    // Detect ON/OFF state change
    IF aUnits[i].bPresVal <> aPrevState[i] THEN
        // --------------------------------------------------------
        // (a) Send TwinCAT message as before
        // --------------------------------------------------------
        IF aUnits[i].bPresVal THEN
            sMsgText := CONCAT(stUnit.sUnitName, ' is Turned ON');
        ELSE
            sMsgText := CONCAT(stUnit.sUnitName, ' is Turned OFF');
        END_IF

        fbMsg.CreateEx(TC_EVENTS.UnitPowerStatus.EventPowerStatus, 0);
        fbMsg.ipArguments.AddString(sMsgText);
        fbMsg.Send(0);

        // --------------------------------------------------------
        // (b) Push event to global CSV queue (for P_CSVWrite_TextMode)
        // --------------------------------------------------------
        IF g_iCount < g_CSV_BUF_SIZE THEN
            g_aUnitName[g_iWriteIdx] := stUnit.sUnitName;
            g_aState[g_iWriteIdx]    := aUnits[i].bPresVal;
            g_iWriteIdx := g_iWriteIdx + 1;
            IF g_iWriteIdx > g_CSV_BUF_SIZE THEN g_iWriteIdx := 1; END_IF
            g_iCount := g_iCount + 1;
        END_IF

        // --------------------------------------------------------
        // (c) Update previous state
        // --------------------------------------------------------
        aPrevState[i] := aUnits[i].bPresVal;
    END_IF
END_FOR

// ------------------------------------------------------------
// Optional debug info
// ------------------------------------------------------------
sDebug := CONCAT('Queued=', INT_TO_STRING(g_iCount));

END_FUNCTION_BLOCK

// ---- POUs/FB_EventLogger/FB_EventF28.TcPOU
FUNCTION_BLOCK FB_EventF28
VAR_INPUT
	FB_Bacnet : FB_BACnet_DAIKIN_MasterStation_III_No_7;
END_VAR
VAR_OUTPUT
	sDebug : STRING(200);
END_VAR
VAR
	fbMsg : FB_TcMessage;
	aUnits : ARRAY[1..23] OF AC_Unit_Status;
	stUnit   : AC_Unit_Status;
	i: INT;
	sMsgText: STRING;

END_VAR
VAR RETAIN
	aPrevState : ARRAY[1..23] OF BOOL := [FALSE(*23*)];
END_VAR


aUnits[1].bPresVal := FB_Bacnet.StartStopStatus_064.bPresVal;
aUnits[1].sUnitName := 'F28-A1 (1-00)';
aUnits[2].bPresVal := FB_Bacnet.StartStopStatus_065.bPresVal;
aUnits[2].sUnitName := 'F28-A2 (1-01)';
aUnits[3].bPresVal := FB_Bacnet.StartStopStatus_066.bPresVal;
aUnits[3].sUnitName := 'F28-A3 (1-02)';
aUnits[4].bPresVal := FB_Bacnet.StartStopStatus_067.bPresVal;
aUnits[4].sUnitName := 'F28-A4 (1-03)';
aUnits[5].bPresVal := FB_Bacnet.StartStopStatus_068.bPresVal;
aUnits[5].sUnitName := 'F28-B1 (1-04)';
aUnits[6].bPresVal := FB_Bacnet.StartStopStatus_069.bPresVal;
aUnits[6].sUnitName := 'F28-B2 (1-05)';
aUnits[7].bPresVal := FB_Bacnet.StartStopStatus_070.bPresVal;
aUnits[7].sUnitName := 'F28-C1 (1-06)';
aUnits[8].bPresVal := FB_Bacnet.StartStopStatus_071.bPresVal;
aUnits[8].sUnitName := 'F28-C2 (1-07)';
aUnits[9].bPresVal := FB_Bacnet.StartStopStatus_072.bPresVal;
aUnits[9].sUnitName := 'F28-D1 (1-08)';
aUnits[10].bPresVal := FB_Bacnet.StartStopStatus_073.bPresVal;
aUnits[10].sUnitName := 'F28-D2 (1-09)';
aUnits[11].bPresVal := FB_Bacnet.StartStopStatus_074.bPresVal;
aUnits[11].sUnitName := 'F28-D3 (1-10)';
aUnits[12].bPresVal := FB_Bacnet.StartStopStatus_075.bPresVal;
aUnits[12].sUnitName := 'F28-D4 (1-11)';
aUnits[13].bPresVal := FB_Bacnet.StartStopStatus_076.bPresVal;
aUnits[13].sUnitName := 'F28-E1 (1-12)';
aUnits[14].bPresVal := FB_Bacnet.StartStopStatus_077.bPresVal;
aUnits[14].sUnitName := 'F28-E2 (1-13)';
aUnits[15].bPresVal := FB_Bacnet.StartStopStatus_078.bPresVal;
aUnits[15].sUnitName := 'F28-E3 (1-14)';
aUnits[16].bPresVal := FB_Bacnet.StartStopStatus_079.bPresVal;
aUnits[16].sUnitName := 'F28-F1 (1-15)';
aUnits[17].bPresVal := FB_Bacnet.StartStopStatus_080.bPresVal;
aUnits[17].sUnitName := 'F28-F2 (2-00)';
aUnits[18].bPresVal := FB_Bacnet.StartStopStatus_081.bPresVal;
aUnits[18].sUnitName := 'F28-G1 (2-01)';
aUnits[19].bPresVal := FB_Bacnet.StartStopStatus_082.bPresVal;
aUnits[19].sUnitName := 'F28-G2 (2-02)';
aUnits[20].bPresVal := FB_Bacnet.StartStopStatus_083.bPresVal;
aUnits[20].sUnitName := 'F28-H (2-03)';
aUnits[21].bPresVal := FB_Bacnet.StartStopStatus_112.bPresVal;
aUnits[21].sUnitName := 'F28-IT-1 (4-00)';
aUnits[22].bPresVal := FB_Bacnet.StartStopStatus_241.bPresVal;
aUnits[22].sUnitName := 'F28-IT-2 (4-01)';
aUnits[23].bPresVal := FB_Bacnet.StartStopStatus_225.bPresVal;
aUnits[23].sUnitName := 'F28-Lobi (3-01)';

FOR i := 1 TO 23 DO
    stUnit := aUnits[i];

    // Detect ON/OFF state change
    IF aUnits[i].bPresVal <> aPrevState[i] THEN
        // --------------------------------------------------------
        // (a) Send TwinCAT message as before
        // --------------------------------------------------------
        IF aUnits[i].bPresVal THEN
            sMsgText := CONCAT(stUnit.sUnitName, ' is Turned ON');
        ELSE
            sMsgText := CONCAT(stUnit.sUnitName, ' is Turned OFF');
        END_IF

        fbMsg.CreateEx(TC_EVENTS.UnitPowerStatus.EventPowerStatus, 0);
        fbMsg.ipArguments.AddString(sMsgText);
        fbMsg.Send(0);

        // --------------------------------------------------------
        // (b) Push event to global CSV queue (for P_CSVWrite_TextMode)
        // --------------------------------------------------------
        IF g_iCount < g_CSV_BUF_SIZE THEN
            g_aUnitName[g_iWriteIdx] := stUnit.sUnitName;
            g_aState[g_iWriteIdx]    := aUnits[i].bPresVal;
            g_iWriteIdx := g_iWriteIdx + 1;
            IF g_iWriteIdx > g_CSV_BUF_SIZE THEN g_iWriteIdx := 1; END_IF
            g_iCount := g_iCount + 1;
        END_IF

        // --------------------------------------------------------
        // (c) Update previous state
        // --------------------------------------------------------
        aPrevState[i] := aUnits[i].bPresVal;
    END_IF
END_FOR

// ------------------------------------------------------------
// Optional debug info
// ------------------------------------------------------------
sDebug := CONCAT('Queued=', INT_TO_STRING(g_iCount));

END_FUNCTION_BLOCK

// ---- POUs/FB_EventLogger/FB_EventF29.TcPOU
FUNCTION_BLOCK FB_EventF29
VAR_INPUT
	FB_Bacnet : FB_BACnet_DAIKIN_MasterStation_III_No_7;
END_VAR
VAR_OUTPUT
	sDebug : STRING(200);
END_VAR
VAR
	fbMsg : FB_TcMessage;
	aUnits : ARRAY[1..23] OF AC_Unit_Status;
	stUnit   : AC_Unit_Status;
	i: INT;
	sMsgText: STRING;

END_VAR
VAR RETAIN
	aPrevState : ARRAY[1..23] OF BOOL := [FALSE(*23*)];
END_VAR


aUnits[1].bPresVal := FB_Bacnet.StartStopStatus_128.bPresVal;
aUnits[1].sUnitName := 'F29-A1 (1-00)';
aUnits[2].bPresVal := FB_Bacnet.StartStopStatus_129.bPresVal;
aUnits[2].sUnitName := 'F29-A2 (1-01)';
aUnits[3].bPresVal := FB_Bacnet.StartStopStatus_130.bPresVal;
aUnits[3].sUnitName := 'F29-A3 (1-02)';
aUnits[4].bPresVal := FB_Bacnet.StartStopStatus_131.bPresVal;
aUnits[4].sUnitName := 'F29-A4 (1-03)';
aUnits[5].bPresVal := FB_Bacnet.StartStopStatus_132.bPresVal;
aUnits[5].sUnitName := 'F29-B1 (1-04)';
aUnits[6].bPresVal := FB_Bacnet.StartStopStatus_133.bPresVal;
aUnits[6].sUnitName := 'F29-B2 (1-05)';
aUnits[7].bPresVal := FB_Bacnet.StartStopStatus_134.bPresVal;
aUnits[7].sUnitName := 'F29-C1 (1-06)';
aUnits[8].bPresVal := FB_Bacnet.StartStopStatus_135.bPresVal;
aUnits[8].sUnitName := 'F29-C2 (1-07)';
aUnits[9].bPresVal := FB_Bacnet.StartStopStatus_136.bPresVal;
aUnits[9].sUnitName := 'F29-D1 (1-08)';
aUnits[10].bPresVal := FB_Bacnet.StartStopStatus_137.bPresVal;
aUnits[10].sUnitName := 'F29-D2 (1-09)';
aUnits[11].bPresVal := FB_Bacnet.StartStopStatus_138.bPresVal;
aUnits[11].sUnitName := 'F29-D3 (1-10)';
aUnits[12].bPresVal := FB_Bacnet.StartStopStatus_139.bPresVal;
aUnits[12].sUnitName := 'F29-D4 (1-11)';
aUnits[13].bPresVal := FB_Bacnet.StartStopStatus_140.bPresVal;
aUnits[13].sUnitName := 'F29-E1 (1-12)';
aUnits[14].bPresVal := FB_Bacnet.StartStopStatus_141.bPresVal;
aUnits[14].sUnitName := 'F29-E2 (1-13)';
aUnits[15].bPresVal := FB_Bacnet.StartStopStatus_142.bPresVal;
aUnits[15].sUnitName := 'F29-E3 (1-14)';
aUnits[16].bPresVal := FB_Bacnet.StartStopStatus_143.bPresVal;
aUnits[16].sUnitName := 'F29-F1 (1-15)';
aUnits[17].bPresVal := FB_Bacnet.StartStopStatus_144.bPresVal;
aUnits[17].sUnitName := 'F29-F2 (2-00)';
aUnits[18].bPresVal := FB_Bacnet.StartStopStatus_145.bPresVal;
aUnits[18].sUnitName := 'F29-G1 (2-01)';
aUnits[19].bPresVal := FB_Bacnet.StartStopStatus_146.bPresVal;
aUnits[19].sUnitName := 'F29-G2 (2-02)';
aUnits[20].bPresVal := FB_Bacnet.StartStopStatus_147.bPresVal;
aUnits[20].sUnitName := 'F29-H (2-03)';
aUnits[21].bPresVal := FB_Bacnet.StartStopStatus_148.bPresVal;
aUnits[21].sUnitName := 'F29-LMR-1 (2-04)';
aUnits[22].bPresVal := FB_Bacnet.StartStopStatus_149.bPresVal;
aUnits[22].sUnitName := 'F29-LMR-2 (2-05)';
aUnits[23].bPresVal := FB_Bacnet.StartStopStatus_226.bPresVal;
aUnits[23].sUnitName := 'F29-Lobi (3-02)';

FOR i := 1 TO 23 DO
    stUnit := aUnits[i];

    // Detect ON/OFF state change
    IF aUnits[i].bPresVal <> aPrevState[i] THEN
        // --------------------------------------------------------
        // (a) Send TwinCAT message as before
        // --------------------------------------------------------
        IF aUnits[i].bPresVal THEN
            sMsgText := CONCAT(stUnit.sUnitName, ' is Turned ON');
        ELSE
            sMsgText := CONCAT(stUnit.sUnitName, ' is Turned OFF');
        END_IF

        fbMsg.CreateEx(TC_EVENTS.UnitPowerStatus.EventPowerStatus, 0);
        fbMsg.ipArguments.AddString(sMsgText);
        fbMsg.Send(0);

        // --------------------------------------------------------
        // (b) Push event to global CSV queue (for P_CSVWrite_TextMode)
        // --------------------------------------------------------
        IF g_iCount < g_CSV_BUF_SIZE THEN
            g_aUnitName[g_iWriteIdx] := stUnit.sUnitName;
            g_aState[g_iWriteIdx]    := aUnits[i].bPresVal;
            g_iWriteIdx := g_iWriteIdx + 1;
            IF g_iWriteIdx > g_CSV_BUF_SIZE THEN g_iWriteIdx := 1; END_IF
            g_iCount := g_iCount + 1;
        END_IF

        // --------------------------------------------------------
        // (c) Update previous state
        // --------------------------------------------------------
        aPrevState[i] := aUnits[i].bPresVal;
    END_IF
END_FOR

// ------------------------------------------------------------
// Optional debug info
// ------------------------------------------------------------
sDebug := CONCAT('Queued=', INT_TO_STRING(g_iCount));

END_FUNCTION_BLOCK

// ---- POUs/FB_EventLogger/FB_EventF30.TcPOU
FUNCTION_BLOCK FB_EventF30
VAR_INPUT
	FB_Bacnet : FB_BACnet_DAIKIN_MasterStation_III_No_7;
END_VAR
VAR_OUTPUT
	sDebug : STRING(200);
END_VAR
VAR
	fbMsg : FB_TcMessage;
	aUnits : ARRAY[1..22] OF AC_Unit_Status;
	stUnit   : AC_Unit_Status;
	i: INT;
	sMsgText: STRING;

END_VAR
VAR RETAIN
	aPrevState : ARRAY[1..22] OF BOOL := [FALSE(*22*)];
END_VAR


aUnits[1].bPresVal := FB_Bacnet.StartStopStatus_192.bPresVal;
aUnits[1].sUnitName := 'F30-A1 (1-00)';
aUnits[2].bPresVal := FB_Bacnet.StartStopStatus_193.bPresVal;
aUnits[2].sUnitName := 'F30-A2 (1-01)';
aUnits[3].bPresVal := FB_Bacnet.StartStopStatus_194.bPresVal;
aUnits[3].sUnitName := 'F30-A3 (1-02)';
aUnits[4].bPresVal := FB_Bacnet.StartStopStatus_195.bPresVal;
aUnits[4].sUnitName := 'F30-B1 (1-03)';
aUnits[5].bPresVal := FB_Bacnet.StartStopStatus_196.bPresVal;
aUnits[5].sUnitName := 'F30-B2 (1-04)';
aUnits[6].bPresVal := FB_Bacnet.StartStopStatus_197.bPresVal;
aUnits[6].sUnitName := 'F30-C1 (1-05)';
aUnits[7].bPresVal := FB_Bacnet.StartStopStatus_198.bPresVal;
aUnits[7].sUnitName := 'F30-C2 (1-06)';
aUnits[8].bPresVal := FB_Bacnet.StartStopStatus_199.bPresVal;
aUnits[8].sUnitName := 'F30-C3 (1-07)';
aUnits[9].bPresVal := FB_Bacnet.StartStopStatus_200.bPresVal;
aUnits[9].sUnitName := 'F30-C4 (1-08)';
aUnits[10].bPresVal := FB_Bacnet.StartStopStatus_201.bPresVal;
aUnits[10].sUnitName := 'F30-C5 (1-09)';
aUnits[11].bPresVal := FB_Bacnet.StartStopStatus_202.bPresVal;
aUnits[11].sUnitName := 'F30-D1 (1-10)';
aUnits[12].bPresVal := FB_Bacnet.StartStopStatus_203.bPresVal;
aUnits[12].sUnitName := 'F30-D2 (1-11)';
aUnits[13].bPresVal := FB_Bacnet.StartStopStatus_204.bPresVal;
aUnits[13].sUnitName := 'F30-D3 (1-12)';
aUnits[14].bPresVal := FB_Bacnet.StartStopStatus_205.bPresVal;
aUnits[14].sUnitName := 'F30-D4 (1-13)';
aUnits[15].bPresVal := FB_Bacnet.StartStopStatus_206.bPresVal;
aUnits[15].sUnitName := 'F30-E1 (1-14)';
aUnits[16].bPresVal := FB_Bacnet.StartStopStatus_207.bPresVal;
aUnits[16].sUnitName := 'F30-E2 (1-15)';
aUnits[17].bPresVal := FB_Bacnet.StartStopStatus_208.bPresVal;
aUnits[17].sUnitName := 'F30-F1 (2-00)';
aUnits[18].bPresVal := FB_Bacnet.StartStopStatus_209.bPresVal;
aUnits[18].sUnitName := 'F30-F2 (2-01)';
aUnits[19].bPresVal := FB_Bacnet.StartStopStatus_210.bPresVal;
aUnits[19].sUnitName := 'F30-G1 (2-02)';
aUnits[20].bPresVal := FB_Bacnet.StartStopStatus_211.bPresVal;
aUnits[20].sUnitName := 'F30-G2 (2-03)';
aUnits[21].bPresVal := FB_Bacnet.StartStopStatus_212.bPresVal;
aUnits[21].sUnitName := 'F30-G3 (2-04)';
aUnits[22].bPresVal := FB_Bacnet.StartStopStatus_227.bPresVal;
aUnits[22].sUnitName := 'F30-Lobi (3-03)';

FOR i := 1 TO 22 DO
    stUnit := aUnits[i];

    // Detect ON/OFF state change
    IF aUnits[i].bPresVal <> aPrevState[i] THEN
        // --------------------------------------------------------
        // (a) Send TwinCAT message as before
        // --------------------------------------------------------
        IF aUnits[i].bPresVal THEN
            sMsgText := CONCAT(stUnit.sUnitName, ' is Turned ON');
        ELSE
            sMsgText := CONCAT(stUnit.sUnitName, ' is Turned OFF');
        END_IF

        fbMsg.CreateEx(TC_EVENTS.UnitPowerStatus.EventPowerStatus, 0);
        fbMsg.ipArguments.AddString(sMsgText);
        fbMsg.Send(0);

        // --------------------------------------------------------
        // (b) Push event to global CSV queue (for P_CSVWrite_TextMode)
        // --------------------------------------------------------
        IF g_iCount < g_CSV_BUF_SIZE THEN
            g_aUnitName[g_iWriteIdx] := stUnit.sUnitName;
            g_aState[g_iWriteIdx]    := aUnits[i].bPresVal;
            g_iWriteIdx := g_iWriteIdx + 1;
            IF g_iWriteIdx > g_CSV_BUF_SIZE THEN g_iWriteIdx := 1; END_IF
            g_iCount := g_iCount + 1;
        END_IF

        // --------------------------------------------------------
        // (c) Update previous state
        // --------------------------------------------------------
        aPrevState[i] := aUnits[i].bPresVal;
    END_IF
END_FOR

// ------------------------------------------------------------
// Optional debug info
// ------------------------------------------------------------
sDebug := CONCAT('Queued=', INT_TO_STRING(g_iCount));

END_FUNCTION_BLOCK

// ---- POUs/FB_EventLogger/FB_EventF31.TcPOU
FUNCTION_BLOCK FB_EventF31
VAR_INPUT
	FB_Bacnet : FB_BACnet_DAIKIN_MasterStation_III_No_8;
END_VAR
VAR_OUTPUT
	sDebug : STRING(200);
END_VAR
VAR
	fbMsg : FB_TcMessage;
	aUnits : ARRAY[1..24] OF AC_Unit_Status;
	stUnit   : AC_Unit_Status;
	i: INT;
	sMsgText: STRING;

END_VAR
VAR RETAIN
	aPrevState : ARRAY[1..24] OF BOOL := [FALSE(*24*)];
END_VAR


aUnits[1].bPresVal := FB_Bacnet.StartStopStatus_000.bPresVal;
aUnits[1].sUnitName := 'F31-A1 (1-00)';
aUnits[2].bPresVal := FB_Bacnet.StartStopStatus_001.bPresVal;
aUnits[2].sUnitName := 'F31-A2 (1-01)';
aUnits[3].bPresVal := FB_Bacnet.StartStopStatus_002.bPresVal;
aUnits[3].sUnitName := 'F31-A3 (1-02)';
aUnits[4].bPresVal := FB_Bacnet.StartStopStatus_003.bPresVal;
aUnits[4].sUnitName := 'F31-B1 (1-03)';
aUnits[5].bPresVal := FB_Bacnet.StartStopStatus_004.bPresVal;
aUnits[5].sUnitName := 'F31-B2 (1-04)';
aUnits[6].bPresVal := FB_Bacnet.StartStopStatus_005.bPresVal;
aUnits[6].sUnitName := 'F31-C1 (1-05)';
aUnits[7].bPresVal := FB_Bacnet.StartStopStatus_006.bPresVal;
aUnits[7].sUnitName := 'F31-C2 (1-06)';
aUnits[8].bPresVal := FB_Bacnet.StartStopStatus_007.bPresVal;
aUnits[8].sUnitName := 'F31-C3 (1-07)';
aUnits[9].bPresVal := FB_Bacnet.StartStopStatus_008.bPresVal;
aUnits[9].sUnitName := 'F31-C4 (1-08)';
aUnits[10].bPresVal := FB_Bacnet.StartStopStatus_009.bPresVal;
aUnits[10].sUnitName := 'F31-C5 (1-09)';
aUnits[11].bPresVal := FB_Bacnet.StartStopStatus_010.bPresVal;
aUnits[11].sUnitName := 'F31-D1 (1-10)';
aUnits[12].bPresVal := FB_Bacnet.StartStopStatus_011.bPresVal;
aUnits[12].sUnitName := 'F31-D2 (1-11)';
aUnits[13].bPresVal := FB_Bacnet.StartStopStatus_012.bPresVal;
aUnits[13].sUnitName := 'F31-D3 (1-12)';
aUnits[14].bPresVal := FB_Bacnet.StartStopStatus_013.bPresVal;
aUnits[14].sUnitName := 'F31-D4 (1-13)';
aUnits[15].bPresVal := FB_Bacnet.StartStopStatus_014.bPresVal;
aUnits[15].sUnitName := 'F31-E1 (1-14)';
aUnits[16].bPresVal := FB_Bacnet.StartStopStatus_015.bPresVal;
aUnits[16].sUnitName := 'F31-E2 (1-15)';
aUnits[17].bPresVal := FB_Bacnet.StartStopStatus_016.bPresVal;
aUnits[17].sUnitName := 'F31-F1 (2-00)';
aUnits[18].bPresVal := FB_Bacnet.StartStopStatus_017.bPresVal;
aUnits[18].sUnitName := 'F31-F2 (2-01)';
aUnits[19].bPresVal := FB_Bacnet.StartStopStatus_018.bPresVal;
aUnits[19].sUnitName := 'F31-G1 (2-02)';
aUnits[20].bPresVal := FB_Bacnet.StartStopStatus_019.bPresVal;
aUnits[20].sUnitName := 'F31-G2 (2-03)';
aUnits[21].bPresVal := FB_Bacnet.StartStopStatus_020.bPresVal;
aUnits[21].sUnitName := 'F31-G3 (2-04)';
//aUnits[22].bPresVal := FB_Bacnet.StartStopStatus_048.bPresVal;
//aUnits[22].sUnitName := 'F31-IT-1 (4-00)';
aUnits[23].bPresVal := FB_Bacnet.StartStopStatus_241.bPresVal;
aUnits[23].sUnitName := 'F31-IT-2 (4-01)';
aUnits[24].bPresVal := FB_Bacnet.StartStopStatus_224.bPresVal;
aUnits[24].sUnitName := 'F31-Lobi (3-00)';

FOR i := 1 TO 24 DO
    stUnit := aUnits[i];

    // Detect ON/OFF state change
    IF aUnits[i].bPresVal <> aPrevState[i] THEN
        // --------------------------------------------------------
        // (a) Send TwinCAT message as before
        // --------------------------------------------------------
        IF aUnits[i].bPresVal THEN
            sMsgText := CONCAT(stUnit.sUnitName, ' is Turned ON');
        ELSE
            sMsgText := CONCAT(stUnit.sUnitName, ' is Turned OFF');
        END_IF

        fbMsg.CreateEx(TC_EVENTS.UnitPowerStatus.EventPowerStatus, 0);
        fbMsg.ipArguments.AddString(sMsgText);
        fbMsg.Send(0);

        // --------------------------------------------------------
        // (b) Push event to global CSV queue (for P_CSVWrite_TextMode)
        // --------------------------------------------------------
        IF g_iCount < g_CSV_BUF_SIZE THEN
            g_aUnitName[g_iWriteIdx] := stUnit.sUnitName;
            g_aState[g_iWriteIdx]    := aUnits[i].bPresVal;
            g_iWriteIdx := g_iWriteIdx + 1;
            IF g_iWriteIdx > g_CSV_BUF_SIZE THEN g_iWriteIdx := 1; END_IF
            g_iCount := g_iCount + 1;
        END_IF

        // --------------------------------------------------------
        // (c) Update previous state
        // --------------------------------------------------------
        aPrevState[i] := aUnits[i].bPresVal;
    END_IF
END_FOR

// ------------------------------------------------------------
// Optional debug info
// ------------------------------------------------------------
sDebug := CONCAT('Queued=', INT_TO_STRING(g_iCount));

END_FUNCTION_BLOCK

// ---- POUs/FB_EventLogger/FB_EventF32.TcPOU
FUNCTION_BLOCK FB_EventF32
VAR_INPUT
	FB_Bacnet : FB_BACnet_DAIKIN_MasterStation_III_No_8;
END_VAR
VAR_OUTPUT
	sDebug : STRING(200);
END_VAR
VAR
	fbMsg : FB_TcMessage;
	aUnits : ARRAY[1..23] OF AC_Unit_Status;
	stUnit   : AC_Unit_Status;
	i: INT;
	sMsgText: STRING;

END_VAR
VAR RETAIN
	aPrevState : ARRAY[1..23] OF BOOL := [FALSE(*23*)];
END_VAR


aUnits[1].bPresVal := FB_Bacnet.StartStopStatus_064.bPresVal;
aUnits[1].sUnitName := 'F32-A1 (1-00)';
aUnits[2].bPresVal := FB_Bacnet.StartStopStatus_065.bPresVal;
aUnits[2].sUnitName := 'F32-A2 (1-01)';
aUnits[3].bPresVal := FB_Bacnet.StartStopStatus_066.bPresVal;
aUnits[3].sUnitName := 'F32-A3 (1-02)';
aUnits[4].bPresVal := FB_Bacnet.StartStopStatus_067.bPresVal;
aUnits[4].sUnitName := 'F32-B1 (1-03)';
aUnits[5].bPresVal := FB_Bacnet.StartStopStatus_068.bPresVal;
aUnits[5].sUnitName := 'F32-B2 (1-04)';
aUnits[6].bPresVal := FB_Bacnet.StartStopStatus_069.bPresVal;
aUnits[6].sUnitName := 'F32-C1 (1-05)';
aUnits[7].bPresVal := FB_Bacnet.StartStopStatus_070.bPresVal;
aUnits[7].sUnitName := 'F32-C2 (1-06)';
aUnits[8].bPresVal := FB_Bacnet.StartStopStatus_071.bPresVal;
aUnits[8].sUnitName := 'F32-C3 (1-07)';
aUnits[9].bPresVal := FB_Bacnet.StartStopStatus_072.bPresVal;
aUnits[9].sUnitName := 'F32-C4 (1-08)';
aUnits[10].bPresVal := FB_Bacnet.StartStopStatus_073.bPresVal;
aUnits[10].sUnitName := 'F32-C5 (1-09)';
aUnits[11].bPresVal := FB_Bacnet.StartStopStatus_074.bPresVal;
aUnits[11].sUnitName := 'F32-D1 (1-10)';
aUnits[12].bPresVal := FB_Bacnet.StartStopStatus_075.bPresVal;
aUnits[12].sUnitName := 'F32-D2 (1-11)';
aUnits[13].bPresVal := FB_Bacnet.StartStopStatus_076.bPresVal;
aUnits[13].sUnitName := 'F32-D3 (1-12)';
aUnits[14].bPresVal := FB_Bacnet.StartStopStatus_077.bPresVal;
aUnits[14].sUnitName := 'F32-D4 (1-13)';
aUnits[15].bPresVal := FB_Bacnet.StartStopStatus_078.bPresVal;
aUnits[15].sUnitName := 'F32-E1 (1-14)';
aUnits[16].bPresVal := FB_Bacnet.StartStopStatus_079.bPresVal;
aUnits[16].sUnitName := 'F32-E2 (1-15)';
aUnits[17].bPresVal := FB_Bacnet.StartStopStatus_080.bPresVal;
aUnits[17].sUnitName := 'F32-F1 (2-00)';
aUnits[18].bPresVal := FB_Bacnet.StartStopStatus_081.bPresVal;
aUnits[18].sUnitName := 'F32-F2 (2-01)';
aUnits[19].bPresVal := FB_Bacnet.StartStopStatus_082.bPresVal;
aUnits[19].sUnitName := 'F32-F3 (2-02)';
aUnits[20].bPresVal := FB_Bacnet.StartStopStatus_083.bPresVal;
aUnits[20].sUnitName := 'F32-F4 (2-03)';
aUnits[21].bPresVal := FB_Bacnet.StartStopStatus_084.bPresVal;
aUnits[21].sUnitName := 'F32-F5 (2-04)';
aUnits[22].bPresVal := FB_Bacnet.StartStopStatus_085.bPresVal;
aUnits[22].sUnitName := 'F32-F6 (2-05)';
aUnits[23].bPresVal := FB_Bacnet.StartStopStatus_225.bPresVal;
aUnits[23].sUnitName := 'F32-Lobi (3-01)';

FOR i := 1 TO 23 DO
    stUnit := aUnits[i];

    // Detect ON/OFF state change
    IF aUnits[i].bPresVal <> aPrevState[i] THEN
        // --------------------------------------------------------
        // (a) Send TwinCAT message as before
        // --------------------------------------------------------
        IF aUnits[i].bPresVal THEN
            sMsgText := CONCAT(stUnit.sUnitName, ' is Turned ON');
        ELSE
            sMsgText := CONCAT(stUnit.sUnitName, ' is Turned OFF');
        END_IF

        fbMsg.CreateEx(TC_EVENTS.UnitPowerStatus.EventPowerStatus, 0);
        fbMsg.ipArguments.AddString(sMsgText);
        fbMsg.Send(0);

        // --------------------------------------------------------
        // (b) Push event to global CSV queue (for P_CSVWrite_TextMode)
        // --------------------------------------------------------
        IF g_iCount < g_CSV_BUF_SIZE THEN
            g_aUnitName[g_iWriteIdx] := stUnit.sUnitName;
            g_aState[g_iWriteIdx]    := aUnits[i].bPresVal;
            g_iWriteIdx := g_iWriteIdx + 1;
            IF g_iWriteIdx > g_CSV_BUF_SIZE THEN g_iWriteIdx := 1; END_IF
            g_iCount := g_iCount + 1;
        END_IF

        // --------------------------------------------------------
        // (c) Update previous state
        // --------------------------------------------------------
        aPrevState[i] := aUnits[i].bPresVal;
    END_IF
END_FOR

// ------------------------------------------------------------
// Optional debug info
// ------------------------------------------------------------
sDebug := CONCAT('Queued=', INT_TO_STRING(g_iCount));

END_FUNCTION_BLOCK

// ---- POUs/FB_EventLogger/FB_EventF33.TcPOU
FUNCTION_BLOCK FB_EventF33
VAR_INPUT
	FB_Bacnet : FB_BACnet_DAIKIN_MasterStation_III_No_8;
END_VAR
VAR_OUTPUT
	sDebug : STRING(200);
END_VAR
VAR
	fbMsg : FB_TcMessage;
	aUnits : ARRAY[1..23] OF AC_Unit_Status;
	stUnit   : AC_Unit_Status;
	i: INT;
	sMsgText: STRING;

END_VAR
VAR RETAIN
	aPrevState : ARRAY[1..23] OF BOOL := [FALSE(*23*)];
END_VAR


aUnits[1].bPresVal := FB_Bacnet.StartStopStatus_128.bPresVal;
aUnits[1].sUnitName := 'F33-A1 (1-00)';
aUnits[2].bPresVal := FB_Bacnet.StartStopStatus_129.bPresVal;
aUnits[2].sUnitName := 'F33-A2 (1-01)';
aUnits[3].bPresVal := FB_Bacnet.StartStopStatus_130.bPresVal;
aUnits[3].sUnitName := 'F33-A3 (1-02)';
aUnits[4].bPresVal := FB_Bacnet.StartStopStatus_131.bPresVal;
aUnits[4].sUnitName := 'F33-B1 (1-03)';
aUnits[5].bPresVal := FB_Bacnet.StartStopStatus_132.bPresVal;
aUnits[5].sUnitName := 'F33-B2 (1-04)';
aUnits[6].bPresVal := FB_Bacnet.StartStopStatus_133.bPresVal;
aUnits[6].sUnitName := 'F33-C1 (1-05)';
aUnits[7].bPresVal := FB_Bacnet.StartStopStatus_134.bPresVal;
aUnits[7].sUnitName := 'F33-C2 (1-06)';
aUnits[8].bPresVal := FB_Bacnet.StartStopStatus_135.bPresVal;
aUnits[8].sUnitName := 'F33-C3 (1-07)';
aUnits[9].bPresVal := FB_Bacnet.StartStopStatus_136.bPresVal;
aUnits[9].sUnitName := 'F33-C4 (1-08)';
aUnits[10].bPresVal := FB_Bacnet.StartStopStatus_137.bPresVal;
aUnits[10].sUnitName := 'F33-C5 (1-09)';
aUnits[11].bPresVal := FB_Bacnet.StartStopStatus_138.bPresVal;
aUnits[11].sUnitName := 'F33-D1 (1-10)';
aUnits[12].bPresVal := FB_Bacnet.StartStopStatus_139.bPresVal;
aUnits[12].sUnitName := 'F33-D2 (1-11)';
aUnits[13].bPresVal := FB_Bacnet.StartStopStatus_140.bPresVal;
aUnits[13].sUnitName := 'F33-D3 (1-12)';
aUnits[14].bPresVal := FB_Bacnet.StartStopStatus_141.bPresVal;
aUnits[14].sUnitName := 'F33-D4 (1-13)';
aUnits[15].bPresVal := FB_Bacnet.StartStopStatus_142.bPresVal;
aUnits[15].sUnitName := 'F33-E1 (1-14)';
aUnits[16].bPresVal := FB_Bacnet.StartStopStatus_143.bPresVal;
aUnits[16].sUnitName := 'F33-E2 (1-15)';
aUnits[17].bPresVal := FB_Bacnet.StartStopStatus_144.bPresVal;
aUnits[17].sUnitName := 'F33-F1 (2-00)';
aUnits[18].bPresVal := FB_Bacnet.StartStopStatus_145.bPresVal;
aUnits[18].sUnitName := 'F33-F2 (2-01)';
aUnits[19].bPresVal := FB_Bacnet.StartStopStatus_146.bPresVal;
aUnits[19].sUnitName := 'F33-F3 (2-02)';
aUnits[20].bPresVal := FB_Bacnet.StartStopStatus_147.bPresVal;
aUnits[20].sUnitName := 'F33-F4 (2-03)';
aUnits[21].bPresVal := FB_Bacnet.StartStopStatus_148.bPresVal;
aUnits[21].sUnitName := 'F33-F5 (2-04)';
aUnits[22].bPresVal := FB_Bacnet.StartStopStatus_149.bPresVal;
aUnits[22].sUnitName := 'F33-F6 (2-05)';
aUnits[23].bPresVal := FB_Bacnet.StartStopStatus_226.bPresVal;
aUnits[23].sUnitName := 'F33-Lobi (3-02)';

FOR i := 1 TO 23 DO
    stUnit := aUnits[i];

    // Detect ON/OFF state change
    IF aUnits[i].bPresVal <> aPrevState[i] THEN
        // --------------------------------------------------------
        // (a) Send TwinCAT message as before
        // --------------------------------------------------------
        IF aUnits[i].bPresVal THEN
            sMsgText := CONCAT(stUnit.sUnitName, ' is Turned ON');
        ELSE
            sMsgText := CONCAT(stUnit.sUnitName, ' is Turned OFF');
        END_IF

        fbMsg.CreateEx(TC_EVENTS.UnitPowerStatus.EventPowerStatus, 0);
        fbMsg.ipArguments.AddString(sMsgText);
        fbMsg.Send(0);

        // --------------------------------------------------------
        // (b) Push event to global CSV queue (for P_CSVWrite_TextMode)
        // --------------------------------------------------------
        IF g_iCount < g_CSV_BUF_SIZE THEN
            g_aUnitName[g_iWriteIdx] := stUnit.sUnitName;
            g_aState[g_iWriteIdx]    := aUnits[i].bPresVal;
            g_iWriteIdx := g_iWriteIdx + 1;
            IF g_iWriteIdx > g_CSV_BUF_SIZE THEN g_iWriteIdx := 1; END_IF
            g_iCount := g_iCount + 1;
        END_IF

        // --------------------------------------------------------
        // (c) Update previous state
        // --------------------------------------------------------
        aPrevState[i] := aUnits[i].bPresVal;
    END_IF
END_FOR

// ------------------------------------------------------------
// Optional debug info
// ------------------------------------------------------------
sDebug := CONCAT('Queued=', INT_TO_STRING(g_iCount));

END_FUNCTION_BLOCK

// ---- POUs/FB_EventLogger/FB_EventF35.TcPOU
FUNCTION_BLOCK FB_EventF35
VAR_INPUT
	FB_Bacnet : FB_BACnet_DAIKIN_MasterStation_III_No_8;
END_VAR
VAR_OUTPUT
	sDebug : STRING(200);
END_VAR
VAR
	fbMsg : FB_TcMessage;
	aUnits : ARRAY[1..25] OF AC_Unit_Status;
	stUnit   : AC_Unit_Status;
	i: INT;
	sMsgText: STRING;

END_VAR
VAR RETAIN
	aPrevState : ARRAY[1..25] OF BOOL := [FALSE(*25*)];
END_VAR


aUnits[1].bPresVal := FB_Bacnet.StartStopStatus_192.bPresVal;
aUnits[1].sUnitName := 'F35-A1 (1-00)';
aUnits[2].bPresVal := FB_Bacnet.StartStopStatus_193.bPresVal;
aUnits[2].sUnitName := 'F35-A2 (1-01)';
aUnits[3].bPresVal := FB_Bacnet.StartStopStatus_194.bPresVal;
aUnits[3].sUnitName := 'F35-A3 (1-02)';
aUnits[4].bPresVal := FB_Bacnet.StartStopStatus_195.bPresVal;
aUnits[4].sUnitName := 'F35-B1 (1-03)';
aUnits[5].bPresVal := FB_Bacnet.StartStopStatus_196.bPresVal;
aUnits[5].sUnitName := 'F35-B2 (1-04)';
aUnits[6].bPresVal := FB_Bacnet.StartStopStatus_197.bPresVal;
aUnits[6].sUnitName := 'F35-C1 (1-05)';
aUnits[7].bPresVal := FB_Bacnet.StartStopStatus_198.bPresVal;
aUnits[7].sUnitName := 'F35-C2 (1-06)';
aUnits[8].bPresVal := FB_Bacnet.StartStopStatus_199.bPresVal;
aUnits[8].sUnitName := 'F35-C3 (1-07)';
aUnits[9].bPresVal := FB_Bacnet.StartStopStatus_200.bPresVal;
aUnits[9].sUnitName := 'F35-C4 (1-08)';
aUnits[10].bPresVal := FB_Bacnet.StartStopStatus_201.bPresVal;
aUnits[10].sUnitName := 'F35-C5 (1-09)';
aUnits[11].bPresVal := FB_Bacnet.StartStopStatus_202.bPresVal;
aUnits[11].sUnitName := 'F35-D1 (1-10)';
aUnits[12].bPresVal := FB_Bacnet.StartStopStatus_203.bPresVal;
aUnits[12].sUnitName := 'F35-D2 (1-11)';
aUnits[13].bPresVal := FB_Bacnet.StartStopStatus_204.bPresVal;
aUnits[13].sUnitName := 'F35-D3 (1-12)';
aUnits[14].bPresVal := FB_Bacnet.StartStopStatus_205.bPresVal;
aUnits[14].sUnitName := 'F35-D4 (1-13)';
aUnits[15].bPresVal := FB_Bacnet.StartStopStatus_206.bPresVal;
aUnits[15].sUnitName := 'F35-E1 (1-14)';
aUnits[16].bPresVal := FB_Bacnet.StartStopStatus_207.bPresVal;
aUnits[16].sUnitName := 'F35-E2 (1-15)';
aUnits[17].bPresVal := FB_Bacnet.StartStopStatus_208.bPresVal;
aUnits[17].sUnitName := 'F35-F1 (2-00)';
aUnits[18].bPresVal := FB_Bacnet.StartStopStatus_209.bPresVal;
aUnits[18].sUnitName := 'F35-F2 (2-01)';
aUnits[19].bPresVal := FB_Bacnet.StartStopStatus_210.bPresVal;
aUnits[19].sUnitName := 'F35-F3 (2-02)';
aUnits[20].bPresVal := FB_Bacnet.StartStopStatus_211.bPresVal;
aUnits[20].sUnitName := 'F35-F4 (2-03)';
aUnits[21].bPresVal := FB_Bacnet.StartStopStatus_212.bPresVal;
aUnits[21].sUnitName := 'F35-F5 (2-04)';
aUnits[22].bPresVal := FB_Bacnet.StartStopStatus_213.bPresVal;
aUnits[22].sUnitName := 'F35-F6 (2-05)';
//aUnits[23].bPresVal := FB_Bacnet.StartStopStatus_242.bPresVal;
//aUnits[23].sUnitName := 'F35-IT-1 (4-02)';
aUnits[24].bPresVal := FB_Bacnet.StartStopStatus_243.bPresVal;
aUnits[24].sUnitName := 'F35-IT-2 (4-03)';
aUnits[25].bPresVal := FB_Bacnet.StartStopStatus_227.bPresVal;
aUnits[25].sUnitName := 'F35-Lobi (3-03)';

FOR i := 1 TO 25 DO
    stUnit := aUnits[i];

    // Detect ON/OFF state change
    IF aUnits[i].bPresVal <> aPrevState[i] THEN
        // --------------------------------------------------------
        // (a) Send TwinCAT message as before
        // --------------------------------------------------------
        IF aUnits[i].bPresVal THEN
            sMsgText := CONCAT(stUnit.sUnitName, ' is Turned ON');
        ELSE
            sMsgText := CONCAT(stUnit.sUnitName, ' is Turned OFF');
        END_IF

        fbMsg.CreateEx(TC_EVENTS.UnitPowerStatus.EventPowerStatus, 0);
        fbMsg.ipArguments.AddString(sMsgText);
        fbMsg.Send(0);

        // --------------------------------------------------------
        // (b) Push event to global CSV queue (for P_CSVWrite_TextMode)
        // --------------------------------------------------------
        IF g_iCount < g_CSV_BUF_SIZE THEN
            g_aUnitName[g_iWriteIdx] := stUnit.sUnitName;
            g_aState[g_iWriteIdx]    := aUnits[i].bPresVal;
            g_iWriteIdx := g_iWriteIdx + 1;
            IF g_iWriteIdx > g_CSV_BUF_SIZE THEN g_iWriteIdx := 1; END_IF
            g_iCount := g_iCount + 1;
        END_IF

        // --------------------------------------------------------
        // (c) Update previous state
        // --------------------------------------------------------
        aPrevState[i] := aUnits[i].bPresVal;
    END_IF
END_FOR

// ------------------------------------------------------------
// Optional debug info
// ------------------------------------------------------------
sDebug := CONCAT('Queued=', INT_TO_STRING(g_iCount));

END_FUNCTION_BLOCK

// ---- POUs/FB_EventLogger/FB_EventF36.TcPOU
FUNCTION_BLOCK FB_EventF36
VAR_INPUT
	FB_Bacnet : FB_BACnet_DAIKIN_MasterStation_III_No_9;
END_VAR
VAR_OUTPUT
	sDebug : STRING(200);
END_VAR
VAR
	fbMsg : FB_TcMessage;
	aUnits : ARRAY[1..23] OF AC_Unit_Status;
	stUnit   : AC_Unit_Status;
	i: INT;
	sMsgText: STRING;

END_VAR
VAR RETAIN
	aPrevState : ARRAY[1..23] OF BOOL := [FALSE(*23*)];
END_VAR


aUnits[1].bPresVal := FB_Bacnet.StartStopStatus_000.bPresVal;
aUnits[1].sUnitName := 'F36-A1 (1-00)';
aUnits[2].bPresVal := FB_Bacnet.StartStopStatus_001.bPresVal;
aUnits[2].sUnitName := 'F36-A2 (1-01)';
aUnits[3].bPresVal := FB_Bacnet.StartStopStatus_002.bPresVal;
aUnits[3].sUnitName := 'F36-A3 (1-02)';
aUnits[4].bPresVal := FB_Bacnet.StartStopStatus_003.bPresVal;
aUnits[4].sUnitName := 'F36-B1 (1-03)';
aUnits[5].bPresVal := FB_Bacnet.StartStopStatus_004.bPresVal;
aUnits[5].sUnitName := 'F36-B2 (1-04)';
aUnits[6].bPresVal := FB_Bacnet.StartStopStatus_005.bPresVal;
aUnits[6].sUnitName := 'F36-C1 (1-05)';
aUnits[7].bPresVal := FB_Bacnet.StartStopStatus_006.bPresVal;
aUnits[7].sUnitName := 'F36-C2 (1-06)';
aUnits[8].bPresVal := FB_Bacnet.StartStopStatus_007.bPresVal;
aUnits[8].sUnitName := 'F36-C3 (1-07)';
aUnits[9].bPresVal := FB_Bacnet.StartStopStatus_008.bPresVal;
aUnits[9].sUnitName := 'F36-C4 (1-08)';
aUnits[10].bPresVal := FB_Bacnet.StartStopStatus_009.bPresVal;
aUnits[10].sUnitName := 'F36-C5 (1-09)';
aUnits[11].bPresVal := FB_Bacnet.StartStopStatus_010.bPresVal;
aUnits[11].sUnitName := 'F36-D1 (1-10)';
aUnits[12].bPresVal := FB_Bacnet.StartStopStatus_011.bPresVal;
aUnits[12].sUnitName := 'F36-D2 (1-11)';
aUnits[13].bPresVal := FB_Bacnet.StartStopStatus_012.bPresVal;
aUnits[13].sUnitName := 'F36-D3 (1-12)';
aUnits[14].bPresVal := FB_Bacnet.StartStopStatus_013.bPresVal;
aUnits[14].sUnitName := 'F36-D4 (1-13)';
aUnits[15].bPresVal := FB_Bacnet.StartStopStatus_014.bPresVal;
aUnits[15].sUnitName := 'F36-E1 (1-14)';
aUnits[16].bPresVal := FB_Bacnet.StartStopStatus_015.bPresVal;
aUnits[16].sUnitName := 'F36-E2 (1-15)';
aUnits[17].bPresVal := FB_Bacnet.StartStopStatus_016.bPresVal;
aUnits[17].sUnitName := 'F36-F1 (2-00)';
aUnits[18].bPresVal := FB_Bacnet.StartStopStatus_017.bPresVal;
aUnits[18].sUnitName := 'F36-F2 (2-01)';
aUnits[19].bPresVal := FB_Bacnet.StartStopStatus_018.bPresVal;
aUnits[19].sUnitName := 'F36-F3 (2-02)';
aUnits[20].bPresVal := FB_Bacnet.StartStopStatus_019.bPresVal;
aUnits[20].sUnitName := 'F36-F4 (2-03)';
aUnits[21].bPresVal := FB_Bacnet.StartStopStatus_020.bPresVal;
aUnits[21].sUnitName := 'F36-F5 (2-04)';
aUnits[22].bPresVal := FB_Bacnet.StartStopStatus_021.bPresVal;
aUnits[22].sUnitName := 'F36-F6 (2-05)';
aUnits[23].bPresVal := FB_Bacnet.StartStopStatus_224.bPresVal;
aUnits[23].sUnitName := 'F36-Lobi (3-00)';

FOR i := 1 TO 23 DO
    stUnit := aUnits[i];

    // Detect ON/OFF state change
    IF aUnits[i].bPresVal <> aPrevState[i] THEN
        // --------------------------------------------------------
        // (a) Send TwinCAT message as before
        // --------------------------------------------------------
        IF aUnits[i].bPresVal THEN
            sMsgText := CONCAT(stUnit.sUnitName, ' is Turned ON');
        ELSE
            sMsgText := CONCAT(stUnit.sUnitName, ' is Turned OFF');
        END_IF

        fbMsg.CreateEx(TC_EVENTS.UnitPowerStatus.EventPowerStatus, 0);
        fbMsg.ipArguments.AddString(sMsgText);
        fbMsg.Send(0);

        // --------------------------------------------------------
        // (b) Push event to global CSV queue (for P_CSVWrite_TextMode)
        // --------------------------------------------------------
        IF g_iCount < g_CSV_BUF_SIZE THEN
            g_aUnitName[g_iWriteIdx] := stUnit.sUnitName;
            g_aState[g_iWriteIdx]    := aUnits[i].bPresVal;
            g_iWriteIdx := g_iWriteIdx + 1;
            IF g_iWriteIdx > g_CSV_BUF_SIZE THEN g_iWriteIdx := 1; END_IF
            g_iCount := g_iCount + 1;
        END_IF

        // --------------------------------------------------------
        // (c) Update previous state
        // --------------------------------------------------------
        aPrevState[i] := aUnits[i].bPresVal;
    END_IF
END_FOR

// ------------------------------------------------------------
// Optional debug info
// ------------------------------------------------------------
sDebug := CONCAT('Queued=', INT_TO_STRING(g_iCount));

END_FUNCTION_BLOCK

// ---- POUs/FB_EventLogger/FB_EventF37.TcPOU
FUNCTION_BLOCK FB_EventF37
VAR_INPUT
	FB_Bacnet : FB_BACnet_DAIKIN_MasterStation_III_No_9;
END_VAR
VAR_OUTPUT
	sDebug : STRING(200);
END_VAR
VAR
	fbMsg : FB_TcMessage;
	aUnits : ARRAY[1..23] OF AC_Unit_Status;
	stUnit   : AC_Unit_Status;
	i: INT;
	sMsgText: STRING;

END_VAR
VAR RETAIN
	aPrevState : ARRAY[1..23] OF BOOL := [FALSE(*23*)];
END_VAR


aUnits[1].bPresVal := FB_Bacnet.StartStopStatus_064.bPresVal;
aUnits[1].sUnitName := 'F37-A1 (1-00)';
aUnits[2].bPresVal := FB_Bacnet.StartStopStatus_065.bPresVal;
aUnits[2].sUnitName := 'F37-A2 (1-01)';
aUnits[3].bPresVal := FB_Bacnet.StartStopStatus_066.bPresVal;
aUnits[3].sUnitName := 'F37-A3 (1-02)';
aUnits[4].bPresVal := FB_Bacnet.StartStopStatus_067.bPresVal;
aUnits[4].sUnitName := 'F37-B1 (1-03)';
aUnits[5].bPresVal := FB_Bacnet.StartStopStatus_068.bPresVal;
aUnits[5].sUnitName := 'F37-B2 (1-04)';
aUnits[6].bPresVal := FB_Bacnet.StartStopStatus_069.bPresVal;
aUnits[6].sUnitName := 'F37-C1 (1-05)';
aUnits[7].bPresVal := FB_Bacnet.StartStopStatus_070.bPresVal;
aUnits[7].sUnitName := 'F37-C2 (1-06)';
aUnits[8].bPresVal := FB_Bacnet.StartStopStatus_071.bPresVal;
aUnits[8].sUnitName := 'F37-C3 (1-07)';
aUnits[9].bPresVal := FB_Bacnet.StartStopStatus_072.bPresVal;
aUnits[9].sUnitName := 'F37-C4 (1-08)';
aUnits[10].bPresVal := FB_Bacnet.StartStopStatus_073.bPresVal;
aUnits[10].sUnitName := 'F37-C5 (1-09)';
aUnits[11].bPresVal := FB_Bacnet.StartStopStatus_074.bPresVal;
aUnits[11].sUnitName := 'F37-D1 (1-10)';
aUnits[12].bPresVal := FB_Bacnet.StartStopStatus_075.bPresVal;
aUnits[12].sUnitName := 'F37-D2 (1-11)';
aUnits[13].bPresVal := FB_Bacnet.StartStopStatus_076.bPresVal;
aUnits[13].sUnitName := 'F37-D3 (1-12)';
aUnits[14].bPresVal := FB_Bacnet.StartStopStatus_077.bPresVal;
aUnits[14].sUnitName := 'F37-D4 (1-13)';
aUnits[15].bPresVal := FB_Bacnet.StartStopStatus_078.bPresVal;
aUnits[15].sUnitName := 'F37-E1 (1-14)';
aUnits[16].bPresVal := FB_Bacnet.StartStopStatus_079.bPresVal;
aUnits[16].sUnitName := 'F37-E2 (1-15)';
aUnits[17].bPresVal := FB_Bacnet.StartStopStatus_080.bPresVal;
aUnits[17].sUnitName := 'F37-F1 (2-00)';
aUnits[18].bPresVal := FB_Bacnet.StartStopStatus_081.bPresVal;
aUnits[18].sUnitName := 'F37-F2 (2-01)';
aUnits[19].bPresVal := FB_Bacnet.StartStopStatus_082.bPresVal;
aUnits[19].sUnitName := 'F37-F3 (2-02)';
aUnits[20].bPresVal := FB_Bacnet.StartStopStatus_083.bPresVal;
aUnits[20].sUnitName := 'F37-F4 (2-03)';
aUnits[21].bPresVal := FB_Bacnet.StartStopStatus_084.bPresVal;
aUnits[21].sUnitName := 'F37-F5 (2-04)';
aUnits[22].bPresVal := FB_Bacnet.StartStopStatus_085.bPresVal;
aUnits[22].sUnitName := 'F37-F6 (2-05)';
aUnits[23].bPresVal := FB_Bacnet.StartStopStatus_225.bPresVal;
aUnits[23].sUnitName := 'F37-Lobi (3-01)';

FOR i := 1 TO 23 DO
    stUnit := aUnits[i];

    // Detect ON/OFF state change
    IF aUnits[i].bPresVal <> aPrevState[i] THEN
        // --------------------------------------------------------
        // (a) Send TwinCAT message as before
        // --------------------------------------------------------
        IF aUnits[i].bPresVal THEN
            sMsgText := CONCAT(stUnit.sUnitName, ' is Turned ON');
        ELSE
            sMsgText := CONCAT(stUnit.sUnitName, ' is Turned OFF');
        END_IF

        fbMsg.CreateEx(TC_EVENTS.UnitPowerStatus.EventPowerStatus, 0);
        fbMsg.ipArguments.AddString(sMsgText);
        fbMsg.Send(0);

        // --------------------------------------------------------
        // (b) Push event to global CSV queue (for P_CSVWrite_TextMode)
        // --------------------------------------------------------
        IF g_iCount < g_CSV_BUF_SIZE THEN
            g_aUnitName[g_iWriteIdx] := stUnit.sUnitName;
            g_aState[g_iWriteIdx]    := aUnits[i].bPresVal;
            g_iWriteIdx := g_iWriteIdx + 1;
            IF g_iWriteIdx > g_CSV_BUF_SIZE THEN g_iWriteIdx := 1; END_IF
            g_iCount := g_iCount + 1;
        END_IF

        // --------------------------------------------------------
        // (c) Update previous state
        // --------------------------------------------------------
        aPrevState[i] := aUnits[i].bPresVal;
    END_IF
END_FOR

// ------------------------------------------------------------
// Optional debug info
// ------------------------------------------------------------
sDebug := CONCAT('Queued=', INT_TO_STRING(g_iCount));

END_FUNCTION_BLOCK

// ---- POUs/FB_EventLogger/FB_EventF38.TcPOU
FUNCTION_BLOCK FB_EventF38
VAR_INPUT
	FB_Bacnet : FB_BACnet_DAIKIN_MasterStation_III_No_9;
END_VAR
VAR_OUTPUT
	sDebug : STRING(200);
END_VAR
VAR
	fbMsg : FB_TcMessage;
	aUnits : ARRAY[1..25] OF AC_Unit_Status;
	stUnit   : AC_Unit_Status;
	i: INT;
	sMsgText: STRING;

END_VAR
VAR RETAIN
	aPrevState : ARRAY[1..25] OF BOOL := [FALSE(*25*)];
END_VAR


aUnits[1].bPresVal := FB_Bacnet.StartStopStatus_128.bPresVal;
aUnits[1].sUnitName := 'F38-A1 (1-00)';
aUnits[2].bPresVal := FB_Bacnet.StartStopStatus_129.bPresVal;
aUnits[2].sUnitName := 'F38-A2 (1-01)';
aUnits[3].bPresVal := FB_Bacnet.StartStopStatus_130.bPresVal;
aUnits[3].sUnitName := 'F38-A3 (1-02)';
aUnits[4].bPresVal := FB_Bacnet.StartStopStatus_131.bPresVal;
aUnits[4].sUnitName := 'F38-B1 (1-03)';
aUnits[5].bPresVal := FB_Bacnet.StartStopStatus_132.bPresVal;
aUnits[5].sUnitName := 'F38-B2 (1-04)';
aUnits[6].bPresVal := FB_Bacnet.StartStopStatus_133.bPresVal;
aUnits[6].sUnitName := 'F38-C1 (1-05)';
aUnits[7].bPresVal := FB_Bacnet.StartStopStatus_134.bPresVal;
aUnits[7].sUnitName := 'F38-C2 (1-06)';
aUnits[8].bPresVal := FB_Bacnet.StartStopStatus_135.bPresVal;
aUnits[8].sUnitName := 'F38-C3 (1-07)';
aUnits[9].bPresVal := FB_Bacnet.StartStopStatus_136.bPresVal;
aUnits[9].sUnitName := 'F38-C4 (1-08)';
aUnits[10].bPresVal := FB_Bacnet.StartStopStatus_137.bPresVal;
aUnits[10].sUnitName := 'F38-C5 (1-09)';
aUnits[11].bPresVal := FB_Bacnet.StartStopStatus_138.bPresVal;
aUnits[11].sUnitName := 'F38-D1 (1-10)';
aUnits[12].bPresVal := FB_Bacnet.StartStopStatus_139.bPresVal;
aUnits[12].sUnitName := 'F38-D2 (1-11)';
aUnits[13].bPresVal := FB_Bacnet.StartStopStatus_140.bPresVal;
aUnits[13].sUnitName := 'F38-D3 (1-12)';
aUnits[14].bPresVal := FB_Bacnet.StartStopStatus_141.bPresVal;
aUnits[14].sUnitName := 'F38-D4 (1-13)';
aUnits[15].bPresVal := FB_Bacnet.StartStopStatus_142.bPresVal;
aUnits[15].sUnitName := 'F38-E1 (1-14)';
aUnits[16].bPresVal := FB_Bacnet.StartStopStatus_143.bPresVal;
aUnits[16].sUnitName := 'F38-E2 (1-15)';
aUnits[17].bPresVal := FB_Bacnet.StartStopStatus_144.bPresVal;
aUnits[17].sUnitName := 'F38-F1 (2-00)';
aUnits[18].bPresVal := FB_Bacnet.StartStopStatus_145.bPresVal;
aUnits[18].sUnitName := 'F38-F2 (2-01)';
aUnits[19].bPresVal := FB_Bacnet.StartStopStatus_146.bPresVal;
aUnits[19].sUnitName := 'F38-F3 (2-02)';
aUnits[20].bPresVal := FB_Bacnet.StartStopStatus_147.bPresVal;
aUnits[20].sUnitName := 'F38-F4 (2-03)';
aUnits[21].bPresVal := FB_Bacnet.StartStopStatus_148.bPresVal;
aUnits[21].sUnitName := 'F38-F5 (2-04)';
aUnits[22].bPresVal := FB_Bacnet.StartStopStatus_149.bPresVal;
aUnits[22].sUnitName := 'F38-F6 (2-05)';
aUnits[23].bPresVal := FB_Bacnet.StartStopStatus_176.bPresVal;
aUnits[23].sUnitName := 'F38-IT-1 (4-00)';
aUnits[24].bPresVal := FB_Bacnet.StartStopStatus_241.bPresVal;
aUnits[24].sUnitName := 'F38-IT-2 (4-01)';
aUnits[25].bPresVal := FB_Bacnet.StartStopStatus_226.bPresVal;
aUnits[25].sUnitName := 'F38-Lobi (3-02)';

FOR i := 1 TO 25 DO
    stUnit := aUnits[i];

    // Detect ON/OFF state change
    IF aUnits[i].bPresVal <> aPrevState[i] THEN
        // --------------------------------------------------------
        // (a) Send TwinCAT message as before
        // --------------------------------------------------------
        IF aUnits[i].bPresVal THEN
            sMsgText := CONCAT(stUnit.sUnitName, ' is Turned ON');
        ELSE
            sMsgText := CONCAT(stUnit.sUnitName, ' is Turned OFF');
        END_IF

        fbMsg.CreateEx(TC_EVENTS.UnitPowerStatus.EventPowerStatus, 0);
        fbMsg.ipArguments.AddString(sMsgText);
        fbMsg.Send(0);

        // --------------------------------------------------------
        // (b) Push event to global CSV queue (for P_CSVWrite_TextMode)
        // --------------------------------------------------------
        IF g_iCount < g_CSV_BUF_SIZE THEN
            g_aUnitName[g_iWriteIdx] := stUnit.sUnitName;
            g_aState[g_iWriteIdx]    := aUnits[i].bPresVal;
            g_iWriteIdx := g_iWriteIdx + 1;
            IF g_iWriteIdx > g_CSV_BUF_SIZE THEN g_iWriteIdx := 1; END_IF
            g_iCount := g_iCount + 1;
        END_IF

        // --------------------------------------------------------
        // (c) Update previous state
        // --------------------------------------------------------
        aPrevState[i] := aUnits[i].bPresVal;
    END_IF
END_FOR

// ------------------------------------------------------------
// Optional debug info
// ------------------------------------------------------------
sDebug := CONCAT('Queued=', INT_TO_STRING(g_iCount));

END_FUNCTION_BLOCK

// ---- POUs/FB_EventLogger/FB_EventF39.TcPOU
FUNCTION_BLOCK FB_EventF39
VAR_INPUT
	FB_Bacnet : FB_BACnet_DAIKIN_MasterStation_III_No_9;
END_VAR
VAR_OUTPUT
	sDebug : STRING(200);
END_VAR
VAR
	fbMsg : FB_TcMessage;
	aUnits : ARRAY[1..23] OF AC_Unit_Status;
	stUnit   : AC_Unit_Status;
	i: INT;
	sMsgText: STRING;

END_VAR
VAR RETAIN
	aPrevState : ARRAY[1..23] OF BOOL := [FALSE(*23*)];
END_VAR


aUnits[1].bPresVal := FB_Bacnet.StartStopStatus_192.bPresVal;
aUnits[1].sUnitName := 'F39-A1 (1-00)';
aUnits[2].bPresVal := FB_Bacnet.StartStopStatus_193.bPresVal;
aUnits[2].sUnitName := 'F39-A2 (1-01)';
aUnits[3].bPresVal := FB_Bacnet.StartStopStatus_194.bPresVal;
aUnits[3].sUnitName := 'F39-A3 (1-02)';
aUnits[4].bPresVal := FB_Bacnet.StartStopStatus_195.bPresVal;
aUnits[4].sUnitName := 'F39-B1 (1-03)';
aUnits[5].bPresVal := FB_Bacnet.StartStopStatus_196.bPresVal;
aUnits[5].sUnitName := 'F39-B2 (1-04)';
aUnits[6].bPresVal := FB_Bacnet.StartStopStatus_197.bPresVal;
aUnits[6].sUnitName := 'F39-C1 (1-05)';
aUnits[7].bPresVal := FB_Bacnet.StartStopStatus_198.bPresVal;
aUnits[7].sUnitName := 'F39-C2 (1-06)';
aUnits[8].bPresVal := FB_Bacnet.StartStopStatus_199.bPresVal;
aUnits[8].sUnitName := 'F39-C3 (1-07)';
aUnits[9].bPresVal := FB_Bacnet.StartStopStatus_200.bPresVal;
aUnits[9].sUnitName := 'F39-C4 (1-08)';
aUnits[10].bPresVal := FB_Bacnet.StartStopStatus_201.bPresVal;
aUnits[10].sUnitName := 'F39-C5 (1-09)';
aUnits[11].bPresVal := FB_Bacnet.StartStopStatus_202.bPresVal;
aUnits[11].sUnitName := 'F39-D1 (1-10)';
aUnits[12].bPresVal := FB_Bacnet.StartStopStatus_203.bPresVal;
aUnits[12].sUnitName := 'F39-D2 (1-11)';
aUnits[13].bPresVal := FB_Bacnet.StartStopStatus_204.bPresVal;
aUnits[13].sUnitName := 'F39-D3 (1-12)';
aUnits[14].bPresVal := FB_Bacnet.StartStopStatus_205.bPresVal;
aUnits[14].sUnitName := 'F39-D4 (1-13)';
aUnits[15].bPresVal := FB_Bacnet.StartStopStatus_206.bPresVal;
aUnits[15].sUnitName := 'F39-E1 (1-14)';
aUnits[16].bPresVal := FB_Bacnet.StartStopStatus_207.bPresVal;
aUnits[16].sUnitName := 'F39-E2 (1-15)';
aUnits[17].bPresVal := FB_Bacnet.StartStopStatus_208.bPresVal;
aUnits[17].sUnitName := 'F39-F1 (2-00)';
aUnits[18].bPresVal := FB_Bacnet.StartStopStatus_209.bPresVal;
aUnits[18].sUnitName := 'F39-F2 (2-01)';
aUnits[19].bPresVal := FB_Bacnet.StartStopStatus_210.bPresVal;
aUnits[19].sUnitName := 'F39-F3 (2-02)';
aUnits[20].bPresVal := FB_Bacnet.StartStopStatus_211.bPresVal;
aUnits[20].sUnitName := 'F39-F4 (2-03)';
aUnits[21].bPresVal := FB_Bacnet.StartStopStatus_212.bPresVal;
aUnits[21].sUnitName := 'F39-F5 (2-04)';
aUnits[22].bPresVal := FB_Bacnet.StartStopStatus_213.bPresVal;
aUnits[22].sUnitName := 'F39-F6 (2-05)';
aUnits[23].bPresVal := FB_Bacnet.StartStopStatus_227.bPresVal;
aUnits[23].sUnitName := 'F39-Lobi (3-03)';

FOR i := 1 TO 23 DO
    stUnit := aUnits[i];

    // Detect ON/OFF state change
    IF aUnits[i].bPresVal <> aPrevState[i] THEN
        // --------------------------------------------------------
        // (a) Send TwinCAT message as before
        // --------------------------------------------------------
        IF aUnits[i].bPresVal THEN
            sMsgText := CONCAT(stUnit.sUnitName, ' is Turned ON');
        ELSE
            sMsgText := CONCAT(stUnit.sUnitName, ' is Turned OFF');
        END_IF

        fbMsg.CreateEx(TC_EVENTS.UnitPowerStatus.EventPowerStatus, 0);
        fbMsg.ipArguments.AddString(sMsgText);
        fbMsg.Send(0);

        // --------------------------------------------------------
        // (b) Push event to global CSV queue (for P_CSVWrite_TextMode)
        // --------------------------------------------------------
        IF g_iCount < g_CSV_BUF_SIZE THEN
            g_aUnitName[g_iWriteIdx] := stUnit.sUnitName;
            g_aState[g_iWriteIdx]    := aUnits[i].bPresVal;
            g_iWriteIdx := g_iWriteIdx + 1;
            IF g_iWriteIdx > g_CSV_BUF_SIZE THEN g_iWriteIdx := 1; END_IF
            g_iCount := g_iCount + 1;
        END_IF

        // --------------------------------------------------------
        // (c) Update previous state
        // --------------------------------------------------------
        aPrevState[i] := aUnits[i].bPresVal;
    END_IF
END_FOR

// ------------------------------------------------------------
// Optional debug info
// ------------------------------------------------------------
sDebug := CONCAT('Queued=', INT_TO_STRING(g_iCount));

END_FUNCTION_BLOCK

// ---- POUs/FB_EventLogger/FB_EventF50.TcPOU
FUNCTION_BLOCK FB_EventF50
VAR_INPUT
	FB_Bacnet : FB_BACnet_DAIKIN_MasterStation_III_No_10;
END_VAR
VAR_OUTPUT
	sDebug : STRING(200);
END_VAR
VAR
	fbMsg : FB_TcMessage;
	aUnits : ARRAY[1..23] OF AC_Unit_Status;
	stUnit   : AC_Unit_Status;
	i: INT;
	sMsgText: STRING;

END_VAR
VAR RETAIN
	aPrevState : ARRAY[1..23] OF BOOL := [FALSE(*23*)];
END_VAR


aUnits[1].bPresVal := FB_Bacnet.StartStopStatus_000.bPresVal;
aUnits[1].sUnitName := 'F50-A1 (1-00)';
aUnits[2].bPresVal := FB_Bacnet.StartStopStatus_001.bPresVal;
aUnits[2].sUnitName := 'F50-A2 (1-01)';
aUnits[3].bPresVal := FB_Bacnet.StartStopStatus_002.bPresVal;
aUnits[3].sUnitName := 'F50-A3 (1-02)';
aUnits[4].bPresVal := FB_Bacnet.StartStopStatus_003.bPresVal;
aUnits[4].sUnitName := 'F50-B1 (1-03)';
aUnits[5].bPresVal := FB_Bacnet.StartStopStatus_004.bPresVal;
aUnits[5].sUnitName := 'F50-B2 (1-04)';
aUnits[6].bPresVal := FB_Bacnet.StartStopStatus_005.bPresVal;
aUnits[6].sUnitName := 'F50-C1 (1-05)';
aUnits[7].bPresVal := FB_Bacnet.StartStopStatus_006.bPresVal;
aUnits[7].sUnitName := 'F50-C2 (1-06)';
aUnits[8].bPresVal := FB_Bacnet.StartStopStatus_007.bPresVal;
aUnits[8].sUnitName := 'F50-C3 (1-07)';
aUnits[9].bPresVal := FB_Bacnet.StartStopStatus_008.bPresVal;
aUnits[9].sUnitName := 'F50-C4 (1-08)';
aUnits[10].bPresVal := FB_Bacnet.StartStopStatus_009.bPresVal;
aUnits[10].sUnitName := 'F50-C5 (1-09)';
aUnits[11].bPresVal := FB_Bacnet.StartStopStatus_010.bPresVal;
aUnits[11].sUnitName := 'F50-D1 (1-10)';
aUnits[12].bPresVal := FB_Bacnet.StartStopStatus_011.bPresVal;
aUnits[12].sUnitName := 'F50-D2 (1-11)';
aUnits[13].bPresVal := FB_Bacnet.StartStopStatus_012.bPresVal;
aUnits[13].sUnitName := 'F50-D3 (1-12)';
aUnits[14].bPresVal := FB_Bacnet.StartStopStatus_013.bPresVal;
aUnits[14].sUnitName := 'F50-D4 (1-13)';
aUnits[15].bPresVal := FB_Bacnet.StartStopStatus_014.bPresVal;
aUnits[15].sUnitName := 'F50-E1 (1-14)';
aUnits[16].bPresVal := FB_Bacnet.StartStopStatus_015.bPresVal;
aUnits[16].sUnitName := 'F50-E2 (1-15)';
aUnits[17].bPresVal := FB_Bacnet.StartStopStatus_016.bPresVal;
aUnits[17].sUnitName := 'F50-F1 (2-00)';
aUnits[18].bPresVal := FB_Bacnet.StartStopStatus_017.bPresVal;
aUnits[18].sUnitName := 'F50-F2 (2-01)';
aUnits[19].bPresVal := FB_Bacnet.StartStopStatus_018.bPresVal;
aUnits[19].sUnitName := 'F50-F3 (2-02)';
aUnits[20].bPresVal := FB_Bacnet.StartStopStatus_019.bPresVal;
aUnits[20].sUnitName := 'F50-F4 (2-03)';
aUnits[21].bPresVal := FB_Bacnet.StartStopStatus_020.bPresVal;
aUnits[21].sUnitName := 'F50-F5 (2-04)';
aUnits[22].bPresVal := FB_Bacnet.StartStopStatus_021.bPresVal;
aUnits[22].sUnitName := 'F50-F6 (2-05)';
aUnits[23].bPresVal := FB_Bacnet.StartStopStatus_234.bPresVal;
aUnits[23].sUnitName := 'F50-Lobi (3-10)';

FOR i := 1 TO 23 DO
    stUnit := aUnits[i];

    // Detect ON/OFF state change
    IF aUnits[i].bPresVal <> aPrevState[i] THEN
        // --------------------------------------------------------
        // (a) Send TwinCAT message as before
        // --------------------------------------------------------
        IF aUnits[i].bPresVal THEN
            sMsgText := CONCAT(stUnit.sUnitName, ' is Turned ON');
        ELSE
            sMsgText := CONCAT(stUnit.sUnitName, ' is Turned OFF');
        END_IF

        fbMsg.CreateEx(TC_EVENTS.UnitPowerStatus.EventPowerStatus, 0);
        fbMsg.ipArguments.AddString(sMsgText);
        fbMsg.Send(0);

        // --------------------------------------------------------
        // (b) Push event to global CSV queue (for P_CSVWrite_TextMode)
        // --------------------------------------------------------
        IF g_iCount < g_CSV_BUF_SIZE THEN
            g_aUnitName[g_iWriteIdx] := stUnit.sUnitName;
            g_aState[g_iWriteIdx]    := aUnits[i].bPresVal;
            g_iWriteIdx := g_iWriteIdx + 1;
            IF g_iWriteIdx > g_CSV_BUF_SIZE THEN g_iWriteIdx := 1; END_IF
            g_iCount := g_iCount + 1;
        END_IF

        // --------------------------------------------------------
        // (c) Update previous state
        // --------------------------------------------------------
        aPrevState[i] := aUnits[i].bPresVal;
    END_IF
END_FOR

// ------------------------------------------------------------
// Optional debug info
// ------------------------------------------------------------
sDebug := CONCAT('Queued=', INT_TO_STRING(g_iCount));

END_FUNCTION_BLOCK

// ---- POUs/FB_EventLogger/FB_EventF51.TcPOU
FUNCTION_BLOCK FB_EventF51
VAR_INPUT
	FB_Bacnet : FB_BACnet_DAIKIN_MasterStation_III_No_10;
END_VAR
VAR_OUTPUT
	sDebug : STRING(200);
END_VAR
VAR
	fbMsg : FB_TcMessage;
	aUnits : ARRAY[1..25] OF AC_Unit_Status;
	stUnit   : AC_Unit_Status;
	i: INT;
	sMsgText: STRING;

END_VAR
VAR RETAIN
	aPrevState : ARRAY[1..25] OF BOOL := [FALSE(*25*)];
END_VAR


aUnits[1].bPresVal := FB_Bacnet.StartStopStatus_064.bPresVal;
aUnits[1].sUnitName := 'F51-A1 (1-00)';
aUnits[2].bPresVal := FB_Bacnet.StartStopStatus_065.bPresVal;
aUnits[2].sUnitName := 'F51-A2 (1-01)';
aUnits[3].bPresVal := FB_Bacnet.StartStopStatus_066.bPresVal;
aUnits[3].sUnitName := 'F51-A3 (1-02)';
aUnits[4].bPresVal := FB_Bacnet.StartStopStatus_067.bPresVal;
aUnits[4].sUnitName := 'F51-B1 (1-03)';
aUnits[5].bPresVal := FB_Bacnet.StartStopStatus_068.bPresVal;
aUnits[5].sUnitName := 'F51-B2 (1-04)';
aUnits[6].bPresVal := FB_Bacnet.StartStopStatus_069.bPresVal;
aUnits[6].sUnitName := 'F51-C1 (1-05)';
aUnits[7].bPresVal := FB_Bacnet.StartStopStatus_070.bPresVal;
aUnits[7].sUnitName := 'F51-C2 (1-06)';
aUnits[8].bPresVal := FB_Bacnet.StartStopStatus_071.bPresVal;
aUnits[8].sUnitName := 'F51-C3 (1-07)';
aUnits[9].bPresVal := FB_Bacnet.StartStopStatus_072.bPresVal;
aUnits[9].sUnitName := 'F51-C4 (1-08)';
aUnits[10].bPresVal := FB_Bacnet.StartStopStatus_073.bPresVal;
aUnits[10].sUnitName := 'F51-C5 (1-09)';
aUnits[11].bPresVal := FB_Bacnet.StartStopStatus_074.bPresVal;
aUnits[11].sUnitName := 'F51-D1 (1-10)';
aUnits[12].bPresVal := FB_Bacnet.StartStopStatus_075.bPresVal;
aUnits[12].sUnitName := 'F51-D2 (1-11)';
aUnits[13].bPresVal := FB_Bacnet.StartStopStatus_076.bPresVal;
aUnits[13].sUnitName := 'F51-D3 (1-12)';
aUnits[14].bPresVal := FB_Bacnet.StartStopStatus_077.bPresVal;
aUnits[14].sUnitName := 'F51-D4 (1-13)';
aUnits[15].bPresVal := FB_Bacnet.StartStopStatus_078.bPresVal;
aUnits[15].sUnitName := 'F51-E1 (1-14)';
aUnits[16].bPresVal := FB_Bacnet.StartStopStatus_079.bPresVal;
aUnits[16].sUnitName := 'F51-E2 (1-15)';
aUnits[17].bPresVal := FB_Bacnet.StartStopStatus_080.bPresVal;
aUnits[17].sUnitName := 'F51-F1 (2-00)';
aUnits[18].bPresVal := FB_Bacnet.StartStopStatus_081.bPresVal;
aUnits[18].sUnitName := 'F51-F2 (2-01)';
aUnits[19].bPresVal := FB_Bacnet.StartStopStatus_082.bPresVal;
aUnits[19].sUnitName := 'F51-F3 (2-02)';
aUnits[20].bPresVal := FB_Bacnet.StartStopStatus_083.bPresVal;
aUnits[20].sUnitName := 'F51-F4 (2-03)';
aUnits[21].bPresVal := FB_Bacnet.StartStopStatus_084.bPresVal;
aUnits[21].sUnitName := 'F51-F5 (2-04)';
aUnits[22].bPresVal := FB_Bacnet.StartStopStatus_085.bPresVal;
aUnits[22].sUnitName := 'F51-F6 (2-05)';
aUnits[23].bPresVal := FB_Bacnet.StartStopStatus_112.bPresVal;
aUnits[23].sUnitName := 'F51-IT-1 (4-00)';
aUnits[24].bPresVal := FB_Bacnet.StartStopStatus_241.bPresVal;
aUnits[24].sUnitName := 'F51-IT-2 (4-01)';
aUnits[25].bPresVal := FB_Bacnet.StartStopStatus_235.bPresVal;
aUnits[25].sUnitName := 'F51-Lobi (3-11)';

FOR i := 1 TO 25 DO
    stUnit := aUnits[i];

    // Detect ON/OFF state change
    IF aUnits[i].bPresVal <> aPrevState[i] THEN
        // --------------------------------------------------------
        // (a) Send TwinCAT message as before
        // --------------------------------------------------------
        IF aUnits[i].bPresVal THEN
            sMsgText := CONCAT(stUnit.sUnitName, ' is Turned ON');
        ELSE
            sMsgText := CONCAT(stUnit.sUnitName, ' is Turned OFF');
        END_IF

        fbMsg.CreateEx(TC_EVENTS.UnitPowerStatus.EventPowerStatus, 0);
        fbMsg.ipArguments.AddString(sMsgText);
        fbMsg.Send(0);

        // --------------------------------------------------------
        // (b) Push event to global CSV queue (for P_CSVWrite_TextMode)
        // --------------------------------------------------------
        IF g_iCount < g_CSV_BUF_SIZE THEN
            g_aUnitName[g_iWriteIdx] := stUnit.sUnitName;
            g_aState[g_iWriteIdx]    := aUnits[i].bPresVal;
            g_iWriteIdx := g_iWriteIdx + 1;
            IF g_iWriteIdx > g_CSV_BUF_SIZE THEN g_iWriteIdx := 1; END_IF
            g_iCount := g_iCount + 1;
        END_IF

        // --------------------------------------------------------
        // (c) Update previous state
        // --------------------------------------------------------
        aPrevState[i] := aUnits[i].bPresVal;
    END_IF
END_FOR

// ------------------------------------------------------------
// Optional debug info
// ------------------------------------------------------------
sDebug := CONCAT('Queued=', INT_TO_STRING(g_iCount));

END_FUNCTION_BLOCK

// ---- POUs/FB_EventLogger/FB_EventF52.TcPOU
FUNCTION_BLOCK FB_EventF52
VAR_INPUT
	FB_Bacnet : FB_BACnet_DAIKIN_MasterStation_III_No_10;
END_VAR
VAR_OUTPUT
	sDebug : STRING(200);
END_VAR
VAR
	fbMsg : FB_TcMessage;
	aUnits : ARRAY[1..23] OF AC_Unit_Status;
	stUnit   : AC_Unit_Status;
	i: INT;
	sMsgText: STRING;

END_VAR
VAR RETAIN
	aPrevState : ARRAY[1..23] OF BOOL := [FALSE(*23*)];
END_VAR


aUnits[1].bPresVal := FB_Bacnet.StartStopStatus_128.bPresVal;
aUnits[1].sUnitName := 'F52-A1 (1-00)';
aUnits[2].bPresVal := FB_Bacnet.StartStopStatus_129.bPresVal;
aUnits[2].sUnitName := 'F52-A2 (1-01)';
aUnits[3].bPresVal := FB_Bacnet.StartStopStatus_130.bPresVal;
aUnits[3].sUnitName := 'F52-A3 (1-02)';
aUnits[4].bPresVal := FB_Bacnet.StartStopStatus_131.bPresVal;
aUnits[4].sUnitName := 'F52-B1 (1-03)';
aUnits[5].bPresVal := FB_Bacnet.StartStopStatus_132.bPresVal;
aUnits[5].sUnitName := 'F52-B2 (1-04)';
aUnits[6].bPresVal := FB_Bacnet.StartStopStatus_133.bPresVal;
aUnits[6].sUnitName := 'F52-C1 (1-05)';
aUnits[7].bPresVal := FB_Bacnet.StartStopStatus_134.bPresVal;
aUnits[7].sUnitName := 'F52-C2 (1-06)';
aUnits[8].bPresVal := FB_Bacnet.StartStopStatus_135.bPresVal;
aUnits[8].sUnitName := 'F52-C3 (1-07)';
aUnits[9].bPresVal := FB_Bacnet.StartStopStatus_136.bPresVal;
aUnits[9].sUnitName := 'F52-C4 (1-08)';
aUnits[10].bPresVal := FB_Bacnet.StartStopStatus_137.bPresVal;
aUnits[10].sUnitName := 'F52-C5 (1-09)';
aUnits[11].bPresVal := FB_Bacnet.StartStopStatus_138.bPresVal;
aUnits[11].sUnitName := 'F52-D1 (1-10)';
aUnits[12].bPresVal := FB_Bacnet.StartStopStatus_139.bPresVal;
aUnits[12].sUnitName := 'F52-D2 (1-11)';
aUnits[13].bPresVal := FB_Bacnet.StartStopStatus_140.bPresVal;
aUnits[13].sUnitName := 'F52-D3 (1-12)';
aUnits[14].bPresVal := FB_Bacnet.StartStopStatus_141.bPresVal;
aUnits[14].sUnitName := 'F52-D4 (1-13)';
aUnits[15].bPresVal := FB_Bacnet.StartStopStatus_142.bPresVal;
aUnits[15].sUnitName := 'F52-E1 (1-14)';
aUnits[16].bPresVal := FB_Bacnet.StartStopStatus_143.bPresVal;
aUnits[16].sUnitName := 'F52-E2 (1-15)';
aUnits[17].bPresVal := FB_Bacnet.StartStopStatus_144.bPresVal;
aUnits[17].sUnitName := 'F52-F1 (2-00)';
aUnits[18].bPresVal := FB_Bacnet.StartStopStatus_145.bPresVal;
aUnits[18].sUnitName := 'F52-F2 (2-01)';
aUnits[19].bPresVal := FB_Bacnet.StartStopStatus_146.bPresVal;
aUnits[19].sUnitName := 'F52-F3 (2-02)';
aUnits[20].bPresVal := FB_Bacnet.StartStopStatus_147.bPresVal;
aUnits[20].sUnitName := 'F52-F4 (2-03)';
aUnits[21].bPresVal := FB_Bacnet.StartStopStatus_148.bPresVal;
aUnits[21].sUnitName := 'F52-F5 (2-04)';
aUnits[22].bPresVal := FB_Bacnet.StartStopStatus_149.bPresVal;
aUnits[22].sUnitName := 'F52-F6 (2-05)';
aUnits[23].bPresVal := FB_Bacnet.StartStopStatus_236.bPresVal;
aUnits[23].sUnitName := 'F52-Lobi (3-12)';

FOR i := 1 TO 23 DO
    stUnit := aUnits[i];

    // Detect ON/OFF state change
    IF aUnits[i].bPresVal <> aPrevState[i] THEN
        // --------------------------------------------------------
        // (a) Send TwinCAT message as before
        // --------------------------------------------------------
        IF aUnits[i].bPresVal THEN
            sMsgText := CONCAT(stUnit.sUnitName, ' is Turned ON');
        ELSE
            sMsgText := CONCAT(stUnit.sUnitName, ' is Turned OFF');
        END_IF

        fbMsg.CreateEx(TC_EVENTS.UnitPowerStatus.EventPowerStatus, 0);
        fbMsg.ipArguments.AddString(sMsgText);
        fbMsg.Send(0);

        // --------------------------------------------------------
        // (b) Push event to global CSV queue (for P_CSVWrite_TextMode)
        // --------------------------------------------------------
        IF g_iCount < g_CSV_BUF_SIZE THEN
            g_aUnitName[g_iWriteIdx] := stUnit.sUnitName;
            g_aState[g_iWriteIdx]    := aUnits[i].bPresVal;
            g_iWriteIdx := g_iWriteIdx + 1;
            IF g_iWriteIdx > g_CSV_BUF_SIZE THEN g_iWriteIdx := 1; END_IF
            g_iCount := g_iCount + 1;
        END_IF

        // --------------------------------------------------------
        // (c) Update previous state
        // --------------------------------------------------------
        aPrevState[i] := aUnits[i].bPresVal;
    END_IF
END_FOR

// ------------------------------------------------------------
// Optional debug info
// ------------------------------------------------------------
sDebug := CONCAT('Queued=', INT_TO_STRING(g_iCount));

END_FUNCTION_BLOCK

// ---- POUs/FB_EventLogger/FB_EventF53.TcPOU
FUNCTION_BLOCK FB_EventF53
VAR_INPUT
	FB_Bacnet : FB_BACnet_DAIKIN_MasterStation_III_No_10;
END_VAR
VAR_OUTPUT
	sDebug : STRING(200);
END_VAR
VAR
	fbMsg : FB_TcMessage;
	aUnits : ARRAY[1..25] OF AC_Unit_Status;
	stUnit   : AC_Unit_Status;
	i: INT;
	sMsgText: STRING;

END_VAR
VAR RETAIN
	aPrevState : ARRAY[1..25] OF BOOL := [FALSE(*25*)];
END_VAR


aUnits[1].bPresVal := FB_Bacnet.StartStopStatus_192.bPresVal;
aUnits[1].sUnitName := 'F53-A1 (1-00)';
aUnits[2].bPresVal := FB_Bacnet.StartStopStatus_193.bPresVal;
aUnits[2].sUnitName := 'F53-A2 (1-01)';
aUnits[3].bPresVal := FB_Bacnet.StartStopStatus_194.bPresVal;
aUnits[3].sUnitName := 'F53-A3 (1-02)';
aUnits[4].bPresVal := FB_Bacnet.StartStopStatus_195.bPresVal;
aUnits[4].sUnitName := 'F53-B1 (1-03)';
aUnits[5].bPresVal := FB_Bacnet.StartStopStatus_196.bPresVal;
aUnits[5].sUnitName := 'F53-B2 (1-04)';
aUnits[6].bPresVal := FB_Bacnet.StartStopStatus_197.bPresVal;
aUnits[6].sUnitName := 'F53-C1 (1-05)';
aUnits[7].bPresVal := FB_Bacnet.StartStopStatus_198.bPresVal;
aUnits[7].sUnitName := 'F53-C2 (1-06)';
aUnits[8].bPresVal := FB_Bacnet.StartStopStatus_199.bPresVal;
aUnits[8].sUnitName := 'F53-C3 (1-07)';
//aUnits[9].bPresVal := FB_Bacnet.StartStopStatus_200.bPresVal;
//aUnits[9].sUnitName := 'F53-C4 (1-08)';
aUnits[10].bPresVal := FB_Bacnet.StartStopStatus_201.bPresVal;
aUnits[10].sUnitName := 'F53-C5 (1-09)';
aUnits[11].bPresVal := FB_Bacnet.StartStopStatus_202.bPresVal;
aUnits[11].sUnitName := 'F53-D1 (1-10)';
aUnits[12].bPresVal := FB_Bacnet.StartStopStatus_203.bPresVal;
aUnits[12].sUnitName := 'F53-D2 (1-11)';
aUnits[13].bPresVal := FB_Bacnet.StartStopStatus_204.bPresVal;
aUnits[13].sUnitName := 'F53-D3 (1-12)';
aUnits[14].bPresVal := FB_Bacnet.StartStopStatus_205.bPresVal;
aUnits[14].sUnitName := 'F53-D4 (1-13)';
aUnits[15].bPresVal := FB_Bacnet.StartStopStatus_206.bPresVal;
aUnits[15].sUnitName := 'F53-E1 (1-14)';
aUnits[16].bPresVal := FB_Bacnet.StartStopStatus_207.bPresVal;
aUnits[16].sUnitName := 'F53-E2 (1-15)';
aUnits[17].bPresVal := FB_Bacnet.StartStopStatus_208.bPresVal;
aUnits[17].sUnitName := 'F53-F1 (2-00)';
aUnits[18].bPresVal := FB_Bacnet.StartStopStatus_209.bPresVal;
aUnits[18].sUnitName := 'F53-F2 (2-01)';
aUnits[19].bPresVal := FB_Bacnet.StartStopStatus_210.bPresVal;
aUnits[19].sUnitName := 'F53-F3 (2-02)';
aUnits[20].bPresVal := FB_Bacnet.StartStopStatus_211.bPresVal;
aUnits[20].sUnitName := 'F53-F4 (2-03)';
aUnits[21].bPresVal := FB_Bacnet.StartStopStatus_212.bPresVal;
aUnits[21].sUnitName := 'F53-F5 (2-04)';
aUnits[22].bPresVal := FB_Bacnet.StartStopStatus_213.bPresVal;
aUnits[22].sUnitName := 'F53-F6 (2-05)';
aUnits[23].bPresVal := FB_Bacnet.StartStopStatus_242.bPresVal;
aUnits[23].sUnitName := 'F53-IT-1 (4-02)';
aUnits[24].bPresVal := FB_Bacnet.StartStopStatus_243.bPresVal;
aUnits[24].sUnitName := 'F53-IT-2 (4-03)';
aUnits[25].bPresVal := FB_Bacnet.StartStopStatus_237.bPresVal;
aUnits[25].sUnitName := 'F53-Lobi (3-13)';

FOR i := 1 TO 25 DO
    stUnit := aUnits[i];

    // Detect ON/OFF state change
    IF aUnits[i].bPresVal <> aPrevState[i] THEN
        // --------------------------------------------------------
        // (a) Send TwinCAT message as before
        // --------------------------------------------------------
        IF aUnits[i].bPresVal THEN
            sMsgText := CONCAT(stUnit.sUnitName, ' is Turned ON');
        ELSE
            sMsgText := CONCAT(stUnit.sUnitName, ' is Turned OFF');
        END_IF

        fbMsg.CreateEx(TC_EVENTS.UnitPowerStatus.EventPowerStatus, 0);
        fbMsg.ipArguments.AddString(sMsgText);
        fbMsg.Send(0);

        // --------------------------------------------------------
        // (b) Push event to global CSV queue (for P_CSVWrite_TextMode)
        // --------------------------------------------------------
        IF g_iCount < g_CSV_BUF_SIZE THEN
            g_aUnitName[g_iWriteIdx] := stUnit.sUnitName;
            g_aState[g_iWriteIdx]    := aUnits[i].bPresVal;
            g_iWriteIdx := g_iWriteIdx + 1;
            IF g_iWriteIdx > g_CSV_BUF_SIZE THEN g_iWriteIdx := 1; END_IF
            g_iCount := g_iCount + 1;
        END_IF

        // --------------------------------------------------------
        // (c) Update previous state
        // --------------------------------------------------------
        aPrevState[i] := aUnits[i].bPresVal;
    END_IF
END_FOR

// ------------------------------------------------------------
// Optional debug info
// ------------------------------------------------------------
sDebug := CONCAT('Queued=', INT_TO_STRING(g_iCount));

END_FUNCTION_BLOCK

// ---- POUs/FB_EventLogger/FB_EventF55.TcPOU
FUNCTION_BLOCK FB_EventF55
VAR_INPUT
	FB_Bacnet : FB_BACnet_DAIKIN_MasterStation_III_No_10;
END_VAR
VAR_OUTPUT
	sDebug : STRING(200);
END_VAR
VAR
	fbMsg : FB_TcMessage;
	aUnits : ARRAY[1..21] OF AC_Unit_Status;
	stUnit   : AC_Unit_Status;
	i: INT;
	sMsgText: STRING;

END_VAR
VAR RETAIN
	aPrevState : ARRAY[1..21] OF BOOL := [FALSE(*21*)];
END_VAR


aUnits[1].bPresVal := FB_Bacnet.StartStopStatus_214.bPresVal;
aUnits[1].sUnitName := 'F55-1 (2-06)';
aUnits[2].bPresVal := FB_Bacnet.StartStopStatus_215.bPresVal;
aUnits[2].sUnitName := 'F55-2 (2-07)';
aUnits[3].bPresVal := FB_Bacnet.StartStopStatus_216.bPresVal;
aUnits[3].sUnitName := 'F55-3 (2-08)';
aUnits[4].bPresVal := FB_Bacnet.StartStopStatus_217.bPresVal;
aUnits[4].sUnitName := 'F55-4 (2-09)';
aUnits[5].bPresVal := FB_Bacnet.StartStopStatus_218.bPresVal;
aUnits[5].sUnitName := 'F55-5 (2-10)';
aUnits[6].bPresVal := FB_Bacnet.StartStopStatus_219.bPresVal;
aUnits[6].sUnitName := 'F55-6 (2-11)';
aUnits[7].bPresVal := FB_Bacnet.StartStopStatus_220.bPresVal;
aUnits[7].sUnitName := 'F55-7 (2-12)';
aUnits[8].bPresVal := FB_Bacnet.StartStopStatus_221.bPresVal;
aUnits[8].sUnitName := 'F55-8 (2-13)';
aUnits[9].bPresVal := FB_Bacnet.StartStopStatus_222.bPresVal;
aUnits[9].sUnitName := 'F55-9 (2-14)';
aUnits[10].bPresVal := FB_Bacnet.StartStopStatus_223.bPresVal;
aUnits[10].sUnitName := 'F55-10 (2-15)';
aUnits[11].bPresVal := FB_Bacnet.StartStopStatus_224.bPresVal;
aUnits[11].sUnitName := 'F55-11 (3-00)';
aUnits[12].bPresVal := FB_Bacnet.StartStopStatus_225.bPresVal;
aUnits[12].sUnitName := 'F55-12 (3-01)';
aUnits[13].bPresVal := FB_Bacnet.StartStopStatus_226.bPresVal;
aUnits[13].sUnitName := 'F55-13 (3-02)';
aUnits[14].bPresVal := FB_Bacnet.StartStopStatus_227.bPresVal;
aUnits[14].sUnitName := 'F55-14 (3-03)';
aUnits[15].bPresVal := FB_Bacnet.StartStopStatus_228.bPresVal;
aUnits[15].sUnitName := 'F55-15 (3-04)';
aUnits[16].bPresVal := FB_Bacnet.StartStopStatus_229.bPresVal;
aUnits[16].sUnitName := 'F55-16 (3-05)';
aUnits[17].bPresVal := FB_Bacnet.StartStopStatus_230.bPresVal;
aUnits[17].sUnitName := 'F55-17 (3-06)';
aUnits[18].bPresVal := FB_Bacnet.StartStopStatus_231.bPresVal;
aUnits[18].sUnitName := 'F55-18 (3-07)';
aUnits[19].bPresVal := FB_Bacnet.StartStopStatus_232.bPresVal;
aUnits[19].sUnitName := 'F55-19 (3-08)';
aUnits[20].bPresVal := FB_Bacnet.StartStopStatus_233.bPresVal;
aUnits[20].sUnitName := 'F55-20 (3-09)';
aUnits[21].bPresVal := FB_Bacnet.StartStopStatus_238.bPresVal;
aUnits[21].sUnitName := 'F55-Lobi (3-14)';

FOR i := 1 TO 21 DO
    stUnit := aUnits[i];

    // Detect ON/OFF state change
    IF aUnits[i].bPresVal <> aPrevState[i] THEN
        // --------------------------------------------------------
        // (a) Send TwinCAT message as before
        // --------------------------------------------------------
        IF aUnits[i].bPresVal THEN
            sMsgText := CONCAT(stUnit.sUnitName, ' is Turned ON');
        ELSE
            sMsgText := CONCAT(stUnit.sUnitName, ' is Turned OFF');
        END_IF

        fbMsg.CreateEx(TC_EVENTS.UnitPowerStatus.EventPowerStatus, 0);
        fbMsg.ipArguments.AddString(sMsgText);
        fbMsg.Send(0);

        // --------------------------------------------------------
        // (b) Push event to global CSV queue (for P_CSVWrite_TextMode)
        // --------------------------------------------------------
        IF g_iCount < g_CSV_BUF_SIZE THEN
            g_aUnitName[g_iWriteIdx] := stUnit.sUnitName;
            g_aState[g_iWriteIdx]    := aUnits[i].bPresVal;
            g_iWriteIdx := g_iWriteIdx + 1;
            IF g_iWriteIdx > g_CSV_BUF_SIZE THEN g_iWriteIdx := 1; END_IF
            g_iCount := g_iCount + 1;
        END_IF

        // --------------------------------------------------------
        // (c) Update previous state
        // --------------------------------------------------------
        aPrevState[i] := aUnits[i].bPresVal;
    END_IF
END_FOR

// ------------------------------------------------------------
// Optional debug info
// ------------------------------------------------------------
sDebug := CONCAT('Queued=', INT_TO_STRING(g_iCount));

END_FUNCTION_BLOCK

// ---- POUs/FB_EventLogger/FB_EventFPH1.TcPOU
FUNCTION_BLOCK FB_EventFPH1
VAR_INPUT
	FB_Bacnet : FB_BACnet_DAIKIN_MasterStation_III_No_10;
END_VAR
VAR_OUTPUT
	sDebug : STRING(200);
END_VAR
VAR
	fbMsg : FB_TcMessage;
	aUnits : ARRAY[1..6] OF AC_Unit_Status;
	stUnit   : AC_Unit_Status;
	i: INT;
	sMsgText: STRING;

END_VAR
VAR RETAIN
	aPrevState : ARRAY[1..6] OF BOOL := [FALSE(*6*)];
END_VAR


aUnits[1].bPresVal := FB_Bacnet.StartStopStatus_150.bPresVal;
aUnits[1].sUnitName := 'FPH1-1 (2-06)';
aUnits[2].bPresVal := FB_Bacnet.StartStopStatus_151.bPresVal;
aUnits[2].sUnitName := 'FPH1-2 (2-07)';
aUnits[3].bPresVal := FB_Bacnet.StartStopStatus_152.bPresVal;
aUnits[3].sUnitName := 'FPH1-3 (2-08)';
aUnits[4].bPresVal := FB_Bacnet.StartStopStatus_153.bPresVal;
aUnits[4].sUnitName := 'FPH1-4 (2-09)';
aUnits[5].bPresVal := FB_Bacnet.StartStopStatus_154.bPresVal;
aUnits[5].sUnitName := 'FPH1-5 (2-10)';
aUnits[6].bPresVal := FB_Bacnet.StartStopStatus_155.bPresVal;
aUnits[6].sUnitName := 'FPH1-6 (2-11)';

FOR i := 1 TO 6 DO
    stUnit := aUnits[i];

    // Detect ON/OFF state change
    IF aUnits[i].bPresVal <> aPrevState[i] THEN
        // --------------------------------------------------------
        // (a) Send TwinCAT message as before
        // --------------------------------------------------------
        IF aUnits[i].bPresVal THEN
            sMsgText := CONCAT(stUnit.sUnitName, ' is Turned ON');
        ELSE
            sMsgText := CONCAT(stUnit.sUnitName, ' is Turned OFF');
        END_IF

        fbMsg.CreateEx(TC_EVENTS.UnitPowerStatus.EventPowerStatus, 0);
        fbMsg.ipArguments.AddString(sMsgText);
        fbMsg.Send(0);

        // --------------------------------------------------------
        // (b) Push event to global CSV queue (for P_CSVWrite_TextMode)
        // --------------------------------------------------------
        IF g_iCount < g_CSV_BUF_SIZE THEN
            g_aUnitName[g_iWriteIdx] := stUnit.sUnitName;
            g_aState[g_iWriteIdx]    := aUnits[i].bPresVal;
            g_iWriteIdx := g_iWriteIdx + 1;
            IF g_iWriteIdx > g_CSV_BUF_SIZE THEN g_iWriteIdx := 1; END_IF
            g_iCount := g_iCount + 1;
        END_IF

        // --------------------------------------------------------
        // (c) Update previous state
        // --------------------------------------------------------
        aPrevState[i] := aUnits[i].bPresVal;
    END_IF
END_FOR

// ------------------------------------------------------------
// Optional debug info
// ------------------------------------------------------------
sDebug := CONCAT('Queued=', INT_TO_STRING(g_iCount));

END_FUNCTION_BLOCK

// ---- POUs/FB_EventLogger/FB_EventFPH2.TcPOU
FUNCTION_BLOCK FB_EventFPH2
VAR_INPUT
	FB_Bacnet : FB_BACnet_DAIKIN_MasterStation_III_No_10;
END_VAR
VAR_OUTPUT
	sDebug : STRING(200);
END_VAR
VAR
	fbMsg : FB_TcMessage;
	aUnits : ARRAY[1..9] OF AC_Unit_Status;
	stUnit   : AC_Unit_Status;
	i: INT;
	sMsgText: STRING;

END_VAR
VAR RETAIN
	aPrevState : ARRAY[1..9] OF BOOL := [FALSE(*9*)];
END_VAR


aUnits[1].bPresVal := FB_Bacnet.StartStopStatus_156.bPresVal;
aUnits[1].sUnitName := 'FPH2-1 (2-12)';
aUnits[2].bPresVal := FB_Bacnet.StartStopStatus_157.bPresVal;
aUnits[2].sUnitName := 'FPH2-2 (2-13)';
aUnits[3].bPresVal := FB_Bacnet.StartStopStatus_158.bPresVal;
aUnits[3].sUnitName := 'FPH2-3 (2-14)';
aUnits[4].bPresVal := FB_Bacnet.StartStopStatus_159.bPresVal;
aUnits[4].sUnitName := 'FPH2-4 (2-15)';
aUnits[5].bPresVal := FB_Bacnet.StartStopStatus_160.bPresVal;
aUnits[5].sUnitName := 'FPH2-5 (3-00)';
aUnits[6].bPresVal := FB_Bacnet.StartStopStatus_161.bPresVal;
aUnits[6].sUnitName := 'FPH2-6 (3-01)';
aUnits[7].bPresVal := FB_Bacnet.StartStopStatus_162.bPresVal;
aUnits[7].sUnitName := 'FPH2-7 (3-02)';
aUnits[8].bPresVal := FB_Bacnet.StartStopStatus_163.bPresVal;
aUnits[8].sUnitName := 'FPH2-8 (3-03)';
aUnits[9].bPresVal := FB_Bacnet.StartStopStatus_164.bPresVal;
aUnits[9].sUnitName := 'FPH2-9 (3-04)';

FOR i := 1 TO 9 DO
    stUnit := aUnits[i];

    // Detect ON/OFF state change
    IF aUnits[i].bPresVal <> aPrevState[i] THEN
        // --------------------------------------------------------
        // (a) Send TwinCAT message as before
        // --------------------------------------------------------
        IF aUnits[i].bPresVal THEN
            sMsgText := CONCAT(stUnit.sUnitName, ' is Turned ON');
        ELSE
            sMsgText := CONCAT(stUnit.sUnitName, ' is Turned OFF');
        END_IF

        fbMsg.CreateEx(TC_EVENTS.UnitPowerStatus.EventPowerStatus, 0);
        fbMsg.ipArguments.AddString(sMsgText);
        fbMsg.Send(0);

        // --------------------------------------------------------
        // (b) Push event to global CSV queue (for P_CSVWrite_TextMode)
        // --------------------------------------------------------
        IF g_iCount < g_CSV_BUF_SIZE THEN
            g_aUnitName[g_iWriteIdx] := stUnit.sUnitName;
            g_aState[g_iWriteIdx]    := aUnits[i].bPresVal;
            g_iWriteIdx := g_iWriteIdx + 1;
            IF g_iWriteIdx > g_CSV_BUF_SIZE THEN g_iWriteIdx := 1; END_IF
            g_iCount := g_iCount + 1;
        END_IF

        // --------------------------------------------------------
        // (c) Update previous state
        // --------------------------------------------------------
        aPrevState[i] := aUnits[i].bPresVal;
    END_IF
END_FOR

// ------------------------------------------------------------
// Optional debug info
// ------------------------------------------------------------
sDebug := CONCAT('Queued=', INT_TO_STRING(g_iCount));

END_FUNCTION_BLOCK

// ---- POUs/FB_EventLogger/FB_EventFPH3.TcPOU
FUNCTION_BLOCK FB_EventFPH3
VAR_INPUT
	FB_Bacnet : FB_BACnet_DAIKIN_MasterStation_III_No_10;
END_VAR
VAR_OUTPUT
	sDebug : STRING(200);
END_VAR
VAR
	fbMsg : FB_TcMessage;
	aUnits : ARRAY[1..9] OF AC_Unit_Status;
	stUnit   : AC_Unit_Status;
	i: INT;
	sMsgText: STRING;

END_VAR
VAR RETAIN
	aPrevState : ARRAY[1..9] OF BOOL := [FALSE(*9*)];
END_VAR


aUnits[1].bPresVal := FB_Bacnet.StartStopStatus_165.bPresVal;
aUnits[1].sUnitName := 'FPH3-1 (3-05)';
aUnits[2].bPresVal := FB_Bacnet.StartStopStatus_166.bPresVal;
aUnits[2].sUnitName := 'FPH3-2 (3-06)';
aUnits[3].bPresVal := FB_Bacnet.StartStopStatus_167.bPresVal;
aUnits[3].sUnitName := 'FPH3-3 (3-07)';
aUnits[4].bPresVal := FB_Bacnet.StartStopStatus_168.bPresVal;
aUnits[4].sUnitName := 'FPH3-4 (3-08)';
aUnits[5].bPresVal := FB_Bacnet.StartStopStatus_169.bPresVal;
aUnits[5].sUnitName := 'FPH3-5 (3-09)';
aUnits[6].bPresVal := FB_Bacnet.StartStopStatus_170.bPresVal;
aUnits[6].sUnitName := 'FPH3-6 (3-10)';
aUnits[7].bPresVal := FB_Bacnet.StartStopStatus_171.bPresVal;
aUnits[7].sUnitName := 'FPH3-7 (3-11)';
aUnits[8].bPresVal := FB_Bacnet.StartStopStatus_172.bPresVal;
aUnits[8].sUnitName := 'FPH3-8 (3-12)';
aUnits[9].bPresVal := FB_Bacnet.StartStopStatus_173.bPresVal;
aUnits[9].sUnitName := 'FPH3-9 (3-13)';

FOR i := 1 TO 9 DO
    stUnit := aUnits[i];

    // Detect ON/OFF state change
    IF aUnits[i].bPresVal <> aPrevState[i] THEN
        // --------------------------------------------------------
        // (a) Send TwinCAT message as before
        // --------------------------------------------------------
        IF aUnits[i].bPresVal THEN
            sMsgText := CONCAT(stUnit.sUnitName, ' is Turned ON');
        ELSE
            sMsgText := CONCAT(stUnit.sUnitName, ' is Turned OFF');
        END_IF

        fbMsg.CreateEx(TC_EVENTS.UnitPowerStatus.EventPowerStatus, 0);
        fbMsg.ipArguments.AddString(sMsgText);
        fbMsg.Send(0);

        // --------------------------------------------------------
        // (b) Push event to global CSV queue (for P_CSVWrite_TextMode)
        // --------------------------------------------------------
        IF g_iCount < g_CSV_BUF_SIZE THEN
            g_aUnitName[g_iWriteIdx] := stUnit.sUnitName;
            g_aState[g_iWriteIdx]    := aUnits[i].bPresVal;
            g_iWriteIdx := g_iWriteIdx + 1;
            IF g_iWriteIdx > g_CSV_BUF_SIZE THEN g_iWriteIdx := 1; END_IF
            g_iCount := g_iCount + 1;
        END_IF

        // --------------------------------------------------------
        // (c) Update previous state
        // --------------------------------------------------------
        aPrevState[i] := aUnits[i].bPresVal;
    END_IF
END_FOR

// ------------------------------------------------------------
// Optional debug info
// ------------------------------------------------------------
sDebug := CONCAT('Queued=', INT_TO_STRING(g_iCount));

END_FUNCTION_BLOCK

// ---- POUs/FB_Scheduler/FB_CurrentTime.TcPOU
FUNCTION_BLOCK FB_CurrentTime
VAR_INPUT
	fbTime   : FB_LocalSystemTime := ( bEnable := TRUE, dwCycle := 1 );
END_VAR
VAR_OUTPUT
END_VAR
VAR
	currH : WORD;
	currM : WORD;
	currD : WORD;
	CurrDate: WORD;
END_VAR

fbTime();
currH := fbTime.systemTime.wHour;
currM := fbTime.systemTime.wMinute;
currD := fbTime.systemTime.wDayOfWeek;
CurrDate := fbTime.systemTime.wDay;

END_FUNCTION_BLOCK

// ---- POUs/FB_Scheduler/FB_Scheduler_FG.TcPOU

      FUNCTION_BLOCK FB_Scheduler_FG
      VAR_INPUT
          currH : WORD;
          currM : WORD;
          currD : WORD;
      END_VAR
      VAR_IN_OUT
          FB_Bacnet : FB_BACnet_DAIKIN_MasterStation_III_No_1;
      END_VAR
      VAR
          i : INT;
          bUnitTriggered : BOOL := FALSE; // New flag to track execution
          prevMinute : WORD := 0;        // New variable to track the previous minute
      END_VAR
      VAR PERSISTENT
          //scheduler var
          bEnSchedFG_ : BOOL := FALSE;
          wSchedWDHourStartFG_ : WORD; 
          wSchedWDMinStartFG_ : WORD; 
          wSchedWEHourStartFG_ : WORD; 
          wSchedWEMinStartFG_ : WORD;
          wSchedWDHourEndFG_ : WORD;
          wSchedWDMinEndFG_ : WORD;
          wSchedWEHourEndFG_ : WORD;
          wSchedWEMinEndFG_ : WORD;
          //unit var
          bUnitFG_ : ARRAY [1..20] OF BOOL;
      END_VAR


        // Reset trigger flag at minute change or at the exact scheduled time
        IF currM <> prevMinute OR 
           (currH = wSchedWDHourStartFG_ AND currM = wSchedWDMinStartFG_) OR 
           (currH = wSchedWDHourEndFG_ AND currM = wSchedWDMinEndFG_) THEN
            bUnitTriggered := FALSE;
            prevMinute := currM;
        END_IF

        // Unit Schedule Enable
        IF bEnSchedFG_ THEN
            // Weekday schedule
            IF currD >= 1 AND currD <= 5 THEN
                IF (wSchedWDHourStartFG_ <> wSchedWDHourEndFG_ OR wSchedWDMinStartFG_ <> wSchedWDMinEndFG_) THEN
                    // Schedule Unit ON
                    IF wSchedWDHourStartFG_ = currH AND wSchedWDMinStartFG_ = currM AND NOT bUnitTriggered THEN
                        bUnitTriggered := TRUE;
                        FOR i := 1 TO 20 DO
                            // Send command unit ON
                            IF bUnitFG_[i] THEN 
                                CASE i OF
                                    1: 
                                        
                                        FB_Bacnet.StartStopCommand_000.bEnWrite := TRUE;
                                        FB_Bacnet.StartStopCommand_000.bVal := TRUE;
                                    2: 
                                        
                                        FB_Bacnet.StartStopCommand_001.bEnWrite := TRUE;
                                        FB_Bacnet.StartStopCommand_001.bVal := TRUE;
                                    3: 
                                        
                                        FB_Bacnet.StartStopCommand_002.bEnWrite := TRUE;
                                        FB_Bacnet.StartStopCommand_002.bVal := TRUE;
                                    4: 
                                        
                                        FB_Bacnet.StartStopCommand_003.bEnWrite := TRUE;
                                        FB_Bacnet.StartStopCommand_003.bVal := TRUE;
                                    5: 
                                        
                                        FB_Bacnet.StartStopCommand_004.bEnWrite := TRUE;
                                        FB_Bacnet.StartStopCommand_004.bVal := TRUE;
                                    6: 
                                        
                                        FB_Bacnet.StartStopCommand_005.bEnWrite := TRUE;
                                        FB_Bacnet.StartStopCommand_005.bVal := TRUE;
                                    7: 
                                        
                                        FB_Bacnet.StartStopCommand_006.bEnWrite := TRUE;
                                        FB_Bacnet.StartStopCommand_006.bVal := TRUE;
                                    8: 
                                        
                                        FB_Bacnet.StartStopCommand_007.bEnWrite := TRUE;
                                        FB_Bacnet.StartStopCommand_007.bVal := TRUE;
                                    9: 
                                        
                                        FB_Bacnet.StartStopCommand_008.bEnWrite := TRUE;
                                        FB_Bacnet.StartStopCommand_008.bVal := TRUE;
                                    10: 
                                        
                                        FB_Bacnet.StartStopCommand_009.bEnWrite := TRUE;
                                        FB_Bacnet.StartStopCommand_009.bVal := TRUE;
                                    11: 
                                        
                                        FB_Bacnet.StartStopCommand_010.bEnWrite := TRUE;
                                        FB_Bacnet.StartStopCommand_010.bVal := TRUE;
                                    12: 
                                        
                                        FB_Bacnet.StartStopCommand_011.bEnWrite := TRUE;
                                        FB_Bacnet.StartStopCommand_011.bVal := TRUE;
                                    13: 
                                        
                                        FB_Bacnet.StartStopCommand_012.bEnWrite := TRUE;
                                        FB_Bacnet.StartStopCommand_012.bVal := TRUE;
                                    14: 
                                        
                                        FB_Bacnet.StartStopCommand_013.bEnWrite := TRUE;
                                        FB_Bacnet.StartStopCommand_013.bVal := TRUE;
                                    15: 
                                        
                                        FB_Bacnet.StartStopCommand_014.bEnWrite := TRUE;
                                        FB_Bacnet.StartStopCommand_014.bVal := TRUE;
                                    16: 
                                        
                                        FB_Bacnet.StartStopCommand_015.bEnWrite := TRUE;
                                        FB_Bacnet.StartStopCommand_015.bVal := TRUE;
                                    17: 
                                        
                                        FB_Bacnet.StartStopCommand_016.bEnWrite := TRUE;
                                        FB_Bacnet.StartStopCommand_016.bVal := TRUE;
                                    18: 
                                        
                                        FB_Bacnet.StartStopCommand_017.bEnWrite := TRUE;
                                        FB_Bacnet.StartStopCommand_017.bVal := TRUE;
                                    19: 
                                        
                                        FB_Bacnet.StartStopCommand_019.bEnWrite := TRUE;
                                        FB_Bacnet.StartStopCommand_019.bVal := TRUE;
                                    20:
                                        
                                        FB_Bacnet.StartStopCommand_018.bEnWrite := TRUE;
                                        FB_Bacnet.StartStopCommand_018.bVal := TRUE;
                                END_CASE
                            END_IF
                        END_FOR
                    END_IF
                    // Schedule Unit OFF
                    IF wSchedWDHourEndFG_ = currH AND wSchedWDMinEndFG_ = currM AND NOT bUnitTriggered THEN
                        bUnitTriggered := TRUE;
                        FOR i := 1 TO 20 DO
                            // Send command unit OFF
                            IF bUnitFG_[i] THEN 
                                CASE i OF
                                    1: 
                                        
                                        FB_Bacnet.StartStopCommand_000.bEnWrite := TRUE;
                                        FB_Bacnet.StartStopCommand_000.bVal := FALSE;
                                    2: 
                                        
                                        FB_Bacnet.StartStopCommand_001.bEnWrite := TRUE;
                                        FB_Bacnet.StartStopCommand_001.bVal := FALSE;
                                    3: 
                                        
                                        FB_Bacnet.StartStopCommand_002.bEnWrite := TRUE;
                                        FB_Bacnet.StartStopCommand_002.bVal := FALSE;
                                    4: 
                                        
                                        FB_Bacnet.StartStopCommand_003.bEnWrite := TRUE;
                                        FB_Bacnet.StartStopCommand_003.bVal := FALSE;
                                    5: 
                                        
                                        FB_Bacnet.StartStopCommand_004.bEnWrite := TRUE;
                                        FB_Bacnet.StartStopCommand_004.bVal := FALSE;
                                    6: 
                                        
                                        FB_Bacnet.StartStopCommand_005.bEnWrite := TRUE;
                                        FB_Bacnet.StartStopCommand_005.bVal := FALSE;
                                    7: 
                                        
                                        FB_Bacnet.StartStopCommand_006.bEnWrite := TRUE;
                                        FB_Bacnet.StartStopCommand_006.bVal := FALSE;
                                    8: 
                                        
                                        FB_Bacnet.StartStopCommand_007.bEnWrite := TRUE;
                                        FB_Bacnet.StartStopCommand_007.bVal := FALSE;
                                    9: 
                                        
                                        FB_Bacnet.StartStopCommand_008.bEnWrite := TRUE;
                                        FB_Bacnet.StartStopCommand_008.bVal := FALSE;
                                    10: 
                                        
                                        FB_Bacnet.StartStopCommand_009.bEnWrite := TRUE;
                                        FB_Bacnet.StartStopCommand_009.bVal := FALSE;
                                    11: 
                                        
                                        FB_Bacnet.StartStopCommand_010.bEnWrite := TRUE;
                                        FB_Bacnet.StartStopCommand_010.bVal := FALSE;
                                    12: 
                                        
                                        FB_Bacnet.StartStopCommand_011.bEnWrite := TRUE;
                                        FB_Bacnet.StartStopCommand_011.bVal := FALSE;
                                    13: 
                                        
                                        FB_Bacnet.StartStopCommand_012.bEnWrite := TRUE;
                                        FB_Bacnet.StartStopCommand_012.bVal := FALSE;
                                    14: 
                                        
                                        FB_Bacnet.StartStopCommand_013.bEnWrite := TRUE;
                                        FB_Bacnet.StartStopCommand_013.bVal := FALSE;
                                    15: 
                                        
                                        FB_Bacnet.StartStopCommand_014.bEnWrite := TRUE;
                                        FB_Bacnet.StartStopCommand_014.bVal := FALSE;
                                    16: 
                                        
                                        FB_Bacnet.StartStopCommand_015.bEnWrite := TRUE;
                                        FB_Bacnet.StartStopCommand_015.bVal := FALSE;
                                    17: 
                                        
                                        FB_Bacnet.StartStopCommand_016.bEnWrite := TRUE;
                                        FB_Bacnet.StartStopCommand_016.bVal := FALSE;
                                    18: 
                                        
                                        FB_Bacnet.StartStopCommand_017.bEnWrite := TRUE;
                                        FB_Bacnet.StartStopCommand_017.bVal := FALSE;
                                    19: 
                                        
                                        FB_Bacnet.StartStopCommand_019.bEnWrite := TRUE;
                                        FB_Bacnet.StartStopCommand_019.bVal := FALSE;
                                    20:
                                        
                                        FB_Bacnet.StartStopCommand_018.bEnWrite := TRUE;
                                        FB_Bacnet.StartStopCommand_018.bVal := FALSE;
                                END_CASE
                            END_IF
                        END_FOR
                    END_IF
                END_IF
            END_IF

            // Weekend schedule
            IF currD = 0 OR currD = 6 THEN
                IF (wSchedWEHourStartFG_ <> wSchedWEHourEndFG_ OR wSchedWEMinStartFG_ <> wSchedWEMinEndFG_) THEN
                    // Schedule Unit ON
                    IF wSchedWEHourStartFG_ = currH AND wSchedWEMinStartFG_ = currM AND NOT bUnitTriggered THEN
                        bUnitTriggered := TRUE;
                        FOR i := 1 TO 20 DO
                            // Send command unit ON
                            IF bUnitFG_[i] THEN 
                                CASE i OF
                                    1: 
                                        
                                        FB_Bacnet.StartStopCommand_000.bEnWrite := TRUE;
                                        FB_Bacnet.StartStopCommand_000.bVal := TRUE;
                                    2: 
                                        
                                        FB_Bacnet.StartStopCommand_001.bEnWrite := TRUE;
                                        FB_Bacnet.StartStopCommand_001.bVal := TRUE;
                                    3: 
                                        
                                        FB_Bacnet.StartStopCommand_002.bEnWrite := TRUE;
                                        FB_Bacnet.StartStopCommand_002.bVal := TRUE;
                                    4: 
                                        
                                        FB_Bacnet.StartStopCommand_003.bEnWrite := TRUE;
                                        FB_Bacnet.StartStopCommand_003.bVal := TRUE;
                                    5: 
                                        
                                        FB_Bacnet.StartStopCommand_004.bEnWrite := TRUE;
                                        FB_Bacnet.StartStopCommand_004.bVal := TRUE;
                                    6: 
                                        
                                        FB_Bacnet.StartStopCommand_005.bEnWrite := TRUE;
                                        FB_Bacnet.StartStopCommand_005.bVal := TRUE;
                                    7: 
                                        
                                        FB_Bacnet.StartStopCommand_006.bEnWrite := TRUE;
                                        FB_Bacnet.StartStopCommand_006.bVal := TRUE;
                                    8: 
                                        
                                        FB_Bacnet.StartStopCommand_007.bEnWrite := TRUE;
                                        FB_Bacnet.StartStopCommand_007.bVal := TRUE;
                                    9: 
                                        
                                        FB_Bacnet.StartStopCommand_008.bEnWrite := TRUE;
                                        FB_Bacnet.StartStopCommand_008.bVal := TRUE;
                                    10: 
                                        
                                        FB_Bacnet.StartStopCommand_009.bEnWrite := TRUE;
                                        FB_Bacnet.StartStopCommand_009.bVal := TRUE;
                                    11: 
                                        
                                        FB_Bacnet.StartStopCommand_010.bEnWrite := TRUE;
                                        FB_Bacnet.StartStopCommand_010.bVal := TRUE;
                                    12: 
                                        
                                        FB_Bacnet.StartStopCommand_011.bEnWrite := TRUE;
                                        FB_Bacnet.StartStopCommand_011.bVal := TRUE;
                                    13: 
                                        
                                        FB_Bacnet.StartStopCommand_012.bEnWrite := TRUE;
                                        FB_Bacnet.StartStopCommand_012.bVal := TRUE;
                                    14: 
                                        
                                        FB_Bacnet.StartStopCommand_013.bEnWrite := TRUE;
                                        FB_Bacnet.StartStopCommand_013.bVal := TRUE;
                                    15: 
                                        
                                        FB_Bacnet.StartStopCommand_014.bEnWrite := TRUE;
                                        FB_Bacnet.StartStopCommand_014.bVal := TRUE;
                                    16: 
                                        
                                        FB_Bacnet.StartStopCommand_015.bEnWrite := TRUE;
                                        FB_Bacnet.StartStopCommand_015.bVal := TRUE;
                                    17: 
                                        
